# B&R Automation Studio project ABC_Pltzr
Automation Studio 4.2.4.149

## Configuration PPC70_24025GEN

CPU 4PPC70.101G-20W, AutomationRuntime D4.22, Build 4.1.2, Vc V4.24.0, Safety 0.0

### Hardware
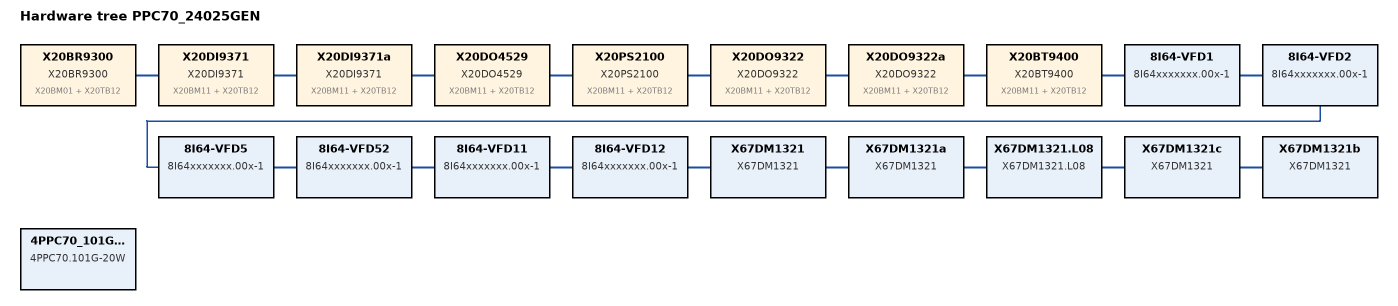
```
4PPC70_101G_20W : 4PPC70.101G-20W v1.2.0.0
  Connector IF1:
    ActivatePowerlink = 0
  Connector IF2:
    ActivateDevice = 1
    Mode = Manual
    InternetAddress = 192.168.1.100
    SubnetMask = 255.255.255.0
    InaNodeNumber = 1
    Vnc1
    VncVcObjectName1 = WSVGA
    VncAuthentication1 = 1
    VncPasswordViewOnly1 = v
    VncPasswordViewControl1 = 24025
    VncMaxConnections1 = 2
    VncRefreshRate1 = 250
  PermanentPvSize = 1000
  RemanentGlobalPvSize = 25000
  VolatileGlobalPvSize = 200000
  EnableUsbRemoteInstall = 1
  TimerDeviceType = SWIOTIMER
  Cyclic1Duration = 4000
  Cyclic1Tolerance = 4000
  Cyclic2Duration = 20000
  Cyclic2Tolerance = 20000
  Cyclic3Duration = 50000
  Cyclic3Tolerance = 50000
  Cyclic4Duration = 100000
  Cyclic4Tolerance = 100000
  Cyclic5Duration = 200000
  Cyclic5Tolerance = 200000
  Cyclic6Duration = 500000
  Cyclic6Tolerance = 500000
  Cyclic7Duration = 1000000
  Cyclic7Tolerance = 1000000
  Cyclic8Duration = 10000
  Cyclic8Tolerance = 30000000
  FtpUser1
  FtpUsername1 = abc
  FtpUserPassword1 = veVz20Da1KUF2Vww53L6omFNdzfk8lHY0HjcrjfOb/w=  // abc123
  FtpUserSalt1 = pyAcjG26
  FTPPath1 = 5
  FTPAccessRight1 = 0
  VcObjectName = WSVGA
  KeyMappingFile = VC\4PPC70_101G_20W.dis
8I64-VFD1 : 8I64xxxxxxx.00x-1 v1.3.8.1  [X2X1 -> X20BT9400.X2X1]
  FunctionModel = Standard
  Supervision = off
  enableIOLR = off
  enableDigitalOutput = off
  DigitalOutputMode01 = actionDO
  ACC = 1
  DEC = 1
  HSP = 900
  ITH = 28
  BFR = 1
  UNS = 460
  FRS = 600
  NCR = 28
  NSP = 1750
  COS = 80
  TFR = 900
  DO = 9
  BRA = 0
  BLC = 64
  BRT = 15
  BEN = 0
  BET = 15
8I64-VFD11 : 8I64xxxxxxx.00x-1 v1.3.8.1  [X2X1 -> 8I64-VFD52.X2X2]
  FunctionModel = Standard
  Supervision = off
  enableIOLR = off
  enableDigitalOutput = off
  DigitalOutputMode01 = actionDO
  DownloadParameters = yes
  ACC = 1
  DEC = 1
  HSP = 900
  ITH = 13
  FTD = 600
  BFR = 1
  UNS = 460
  FRS = 600
  NCR = 13
  NSP = 1750
  COS = 80
  TFR = 900
  DO = 9
  BRA = 0
  BLC = 64
  BRT = 5
  BEN = 0
  BET = 5
8I64-VFD12 : 8I64xxxxxxx.00x-1 v1.3.8.1  [X2X1 -> 8I64-VFD11.X2X2]
  FunctionModel = Standard
  Supervision = off
  enableIOLR = off
  enableDigitalOutput = off
  DigitalOutputMode01 = actionDO
  DownloadParameters = yes
  ACC = 1
  DEC = 200
  HSP = 900
  ITH = 13
  FTD = 600
  BFR = 1
  UNS = 460
  FRS = 600
  NCR = 13
  NSP = 1750
  COS = 80
  TFR = 900
  DO = 9
  BRA = 0
  BLC = 64
  BRT = 5
  BEN = 0
  BET = 5
8I64-VFD2 : 8I64xxxxxxx.00x-1 v1.3.8.1  [X2X1 -> 8I64-VFD1.X2X2]
  FunctionModel = Standard
  Supervision = off
  enableIOLR = off
  enableDigitalOutput = off
  DigitalOutputMode01 = actionDO
  DownloadParameters = yes
  ACC = 1
  DEC = 1
  HSP = 900
  BFR = 1
  UNS = 460
  FRS = 600
  NCR = 13
  NSP = 1750
  TFR = 900
  DO = 9
  BRA = 0
  BLC = 64
  BRT = 5
  BEN = 0
  BET = 5
8I64-VFD5 : 8I64xxxxxxx.00x-1 v1.3.8.1  [X2X1 -> 8I64-VFD2.X2X2]
  FunctionModel = Standard
  Supervision = off
  DownloadParameters = yes
  ACC = 1
  DEC = 1
  HSP = 900
  ITH = 13
  FTD = 600
  BFR = 1
  UNS = 460
  FRS = 600
  NCR = 13
  NSP = 1750
  COS = 80
  TFR = 900
  DE2 = 10
  BRA = 0
8I64-VFD52 : 8I64xxxxxxx.00x-1 v1.3.8.1  [X2X1 -> 8I64-VFD5.X2X2]
  FunctionModel = Standard
  Supervision = off
  enableIOLR = off
  enableDigitalOutput = off
  DigitalOutputMode01 = actionDO
  ACC = 1
  DEC = 1
  HSP = 900
  ITH = 13
  FTD = 600
  BFR = 1
  UNS = 460
  FRS = 600
  NCR = 13
  NSP = 1750
  COS = 80
  TFR = 900
  DO = 9
  INR = 0
  BRA = 0
  BLC = 64
  BRT = 1
  BEN = 0
  BET = 1
X20BM01 : X20BM01 v1.0.0.1
X20BM11 : X20BM11 v1.0.0.0  [X2X1 -> X20BM01.X2X2]
X20BM11a : X20BM11 v1.0.0.0  [X2X1 -> X20BM11.X2X2]
X20BM11b : X20BM11 v1.0.0.0  [X2X1 -> X20BM11a.X2X2]
X20BM11c : X20BM11 v1.0.0.0  [X2X1 -> X20BM11b.X2X2]
X20BM11d : X20BM11 v1.0.0.0  [X2X1 -> X20BM11c.X2X2]
X20BM11e : X20BM11 v1.0.0.0  [X2X1 -> X20BM11f.X2X2]
X20BM11f : X20BM11 v1.0.0.0  [X2X1 -> X20BM11d.X2X2]
X20BR9300 : X20BR9300 v1.0.2.6  [SS1 -> X20TB12.SS; SL -> X20BM01.SL1; X2X1 -> 4PPC70_101G_20W.IF5]
  Supervision = off
X20BT9400 : X20BT9400 v1.0.1.3  [SS1 -> X20TB12f.SS; SL -> X20BM11e.SL1]
  Supervision = off
X20DI9371 : X20DI9371 v1.0.1.2  [SS1 -> X20TB12a.SS; SL -> X20BM11.SL1]
  Supervision = off
X20DI9371a : X20DI9371 v1.0.1.2  [SS1 -> X20TB12b.SS; SL -> X20BM11a.SL1]
  Supervision = off
  InputFilter = 100
X20DO4529 : X20DO4529 v1.0.1.2  [SS1 -> X20TB12c.SS; SL -> X20BM11b.SL1]
  Supervision = off
X20DO9322 : X20DO9322 v1.0.3.0  [SS1 -> X20TB12e.SS; SL -> X20BM11d.SL1]
  Supervision = off
X20DO9322a : X20DO9322 v1.0.3.0  [SS1 -> X20TB12g.SS; SL -> X20BM11f.SL1]
  Supervision = off
X20PS2100 : X20PS2100 v1.0.3.0  [SS1 -> X20TB12d.SS; SL -> X20BM11c.SL1]
  Supervision = off
X20TB12 : X20TB12 v1.0.0.0
X20TB12a : X20TB12 v1.0.0.0
X20TB12b : X20TB12 v1.0.0.0
X20TB12c : X20TB12 v1.0.0.0
X20TB12d : X20TB12 v1.0.0.0
X20TB12e : X20TB12 v1.0.0.0
X20TB12f : X20TB12 v1.0.0.0
X20TB12g : X20TB12 v1.0.0.0
X67DM1321 : X67DM1321 v1.1.1.0  [X2X1 -> 8I64-VFD12.X2X2]
  Supervision = off
X67DM1321.L08 : X67DM1321.L08 v1.1.2.0  [X2X1 -> X67DM1321a.X2X2]
  Supervision = off
  Direction01 = output
  Direction02 = output
  Direction03 = output
  Direction04 = output
  Direction05 = output
  Direction06 = output
  Direction07 = output
  Direction08 = output
  Direction09 = output
  Direction10 = output
  Direction11 = output
  Direction12 = output
X67DM1321a : X67DM1321 v1.1.1.0  [X2X1 -> X67DM1321.X2X2]
  Supervision = off
  Direction01 = output
  Direction02 = output
  Direction03 = output
  Direction04 = output
X67DM1321b : X67DM1321 v1.1.1.0  [X2X1 -> X67DM1321c.X2X2]
  Supervision = off
X67DM1321c : X67DM1321 v1.1.1.0  [X2X1 -> X67DM1321.L08.X2X2]
  Supervision = off
  Direction01 = output
  Direction02 = output
```

## Configuration PPC70_JOB24025

### Task classes (Cpu.sw)
```
Cyclic#1:
  diofilter <- MachineControl.diofilter.prg
  simonly <- MachineControl.simonly.prg
  alarms <- MachineControl.alarms.prg
  messages <- MachineControl.messages.prg
  machCtrl <- MachineControl.machCtrl.prg
  machzero <- MachineControl.machzero.prg
  vfdControl <- MachineControl.vfdControl.prg
  safety <- MachineControl.safety.prg
  counter <- Simulation.counter.prg
  machmode <- MachineControl.machmode.prg
  caseturner <- MachineControl.caseturner.prg
  blades <- MachineControl.blades.prg
  rowforming <- MachineControl.rowforming.prg
  transtable <- MachineControl.transtable.prg
  retainbar <- MachineControl.retainbar.prg
  squaring <- MachineControl.squaring.prg
  elevator <- MachineControl.elevator.prg
  elevmove <- MachineControl.elevmove.prg
  palletinfe <- MachineControl.palletinfcv.prg
  palletdisc <- MachineControl.palletdischarge.prg
  infcvidle <- MachineControl.infcvidle.prg
  palletinfa <- MachineControl.palletinfauto.prg [disabled]
  animation <- MachineControl.animation.prg [disabled]
  palProc <- MachineControl.palProc.prg
  drycycle <- MachineControl.drycycle.prg [disabled]
  drycypal <- MachineControl.drycypal.prg [disabled]
Cyclic#4:
  X64param <- ParameterDownload.X64_S44_Download.X64param.prg [disabled]
  paiVFDX64 <- paiComponents.paiBnRVFD.paiVFDX64.prg
Cyclic#8:
  paiHmi <- paiComponents.paiTemplate.paiHMI.paiHmi.prg
  paiFS <- paiComponents.paiFileService.paiFS.prg
  paiMp <- paiComponents.paiMp.paiMp.prg
  paiFileDT <- paiComponents.paiMp.paiFileDT.prg
  paiUser <- paiComponents.paiUser.paiUser.prg
  appHmi <- MachineControl.appHmi.prg
  appDraw <- MachineControl.appDraw.prg
  appCfgRec <- appConfigAndRecipes.appCfgRec.prg
  paiPingSer <- paiComponents.paiPing.paiPingService.prg
  read_data <- paiComponents.LibAsUSB1_ST.read_data.prg [disabled]
VcDataObjects: WSVGA <- HMI.WSVGA.dob
Binaries: vccdt, vccbmp, vccline, vcfile, arial, vctcal, WSVGA02, vcrt, vcmgr, vccstr, vcbclass, vccbtn, vcgclass, vcdsint, vcchtml, vccpwd, vcshared, vccddbox, vccscale, arialbd, vcxml, vccnum, vccalarm, visvc, vccurl, vccslider, vcctext, vcpdsw, vcfntttf, vccovl, vccshape, ariblk, cour, vcctrend, vcclbox, vccpopup, vcdsloc, vcchspot, vcalarm, WSVGA01, WSVGA03, vcpdvnc, vcpkat, vcnet, vccdbox, vcpdi815, vcptelo, vcpdihd, vcpdi855, vcpfppc7, vcpk, Config_4, Config_3, Config_1, iomap, ashwd, Config_2, asfw, Config, arconfig, sysconf, vcpfar00
Libraries: sprintf2, bgringbuf, bglibas, standard, AsIecCon, Operator, asstring, brsystem, sys_lib, AsARCfg, AsUPS, FileIO, AsICMP, AsBrStr, MpCom, MpFile, MpRecipe, MpAlarm, dvframe, astime, visapi, arsvcreg, vcresman, dataobj, AsIOAcc, runtime, AsMem, AsMath, AsEPL, CSV_File, AsUSB
```

### Config_2.mpalarmbasic - 4PPC70_101G_20F005/mapp/Config_2.mpalarmbasic
```
Element gMpLinkMpAlarmBasic (Type=mpalarmbasic)
  mapp.Alarm.Factory:
    Reactions:
      Reaction[0]:
        Description = Example: Immediate Stop
  Alarms:
    UserAlarm:
      Alarms:
        Alarm[0]:
          ID = 0
          Description = Example: Temperature over Tolerance
          Reaction = 1
```

### Config_3.mprecipexml - 4PPC70_101G_20F005/mapp/Config_3.mprecipexml
```
Element gMpLinkMpRecipeXmlCustom1 (Type=mprecipexml)
```

## Configuration PPC70_Ver1

CPU 4PPC70.101G-20F005, AutomationRuntime D4.22, Build 4.1.2, Vc V4.22.0

### Task classes (Cpu.sw)
```
Cyclic#1:
  simonly <- MachineControl.simonly.prg
  alarms <- MachineControl.alarms.prg
  messages <- MachineControl.messages.prg
  machCtrl <- MachineControl.machCtrl.prg
  machzero <- MachineControl.machzero.prg
  vfdControl <- MachineControl.vfdControl.prg
  safety <- MachineControl.safety.prg
  counter <- Simulation.counter.prg
  machmode <- MachineControl.machmode.prg
  caseturner <- MachineControl.caseturner.prg
  blades <- MachineControl.blades.prg
  rowforming <- MachineControl.rowforming.prg
  transtable <- MachineControl.transtable.prg
  retainbar <- MachineControl.retainbar.prg
  squaring <- MachineControl.squaring.prg
  elevator <- MachineControl.elevator.prg
  elevmove <- MachineControl.elevmove.prg
  palletinfe <- MachineControl.palletinfcv.prg
  palletdisc <- MachineControl.palletdischarge.prg
  palletinfa <- MachineControl.palletinfauto.prg
  animation <- MachineControl.animation.prg [disabled]
  palProc <- MachineControl.palProc.prg
  drycycle <- MachineControl.drycycle.prg [disabled]
  drycypal <- MachineControl.drycypal.prg [disabled]
Cyclic#4:
  X64param <- ParameterDownload.X64_S44_Download.X64param.prg [disabled]
Cyclic#8:
  paiHmi <- paiComponents.paiTemplate.paiHMI.paiHmi.prg
  paiFS <- paiComponents.paiFileService.paiFS.prg
  paiMp <- paiComponents.paiMp.paiMp.prg
  paiFileDT <- paiComponents.paiMp.paiFileDT.prg
  paiUser <- paiComponents.paiUser.paiUser.prg
  appHmi <- MachineControl.appHmi.prg
  appDraw <- MachineControl.appDraw.prg
  appCfgRec <- appConfigAndRecipes.appCfgRec.prg
  paiPingSer <- paiComponents.paiPing.paiPingService.prg
VcDataObjects: WSVGA <- HMI.WSVGA.dob
Binaries: vccdt, vccbmp, vccline, vcfile, arial, vctcal, WSVGA02, vcrt, vcmgr, vccstr, vcbclass, vccbtn, vcgclass, vcdsint, vcchtml, vccpwd, vcshared, vccddbox, vccscale, arialbd, vcxml, vccnum, vccalarm, visvc, vccurl, vccslider, vcctext, vcpdsw, vcfntttf, vccovl, vccshape, ariblk, cour, vcctrend, vcclbox, vccpopup, vcdsloc, vcchspot, vcalarm, WSVGA01, WSVGA03, vcpdvnc, vcpkat, vcnet, vccdbox, vcpk, vcpfppc7, vcpdi855, vcpdihd, vcptelo, vcpdi815, vcpfar00, Config_4, Config_3, Config_1, iomap, ashwd, Config_2, asfw, Config, arconfig, sysconf
Libraries: sprintf2, bgringbuf, bglibas, standard, AsIecCon, Operator, asstring, brsystem, sys_lib, AsARCfg, AsUPS, FileIO, AsICMP, AsBrStr, MpCom, MpFile, MpRecipe, MpAlarm, dvframe, astime, visapi, arsvcreg, vcresman, dataobj, AsIOAcc, runtime, AsMem, AsMath, AsEPL, CSV_File
```

### IoMap.iom - 4PPC70_101G_20F005/IoMap.iom
```iecst
(*********************************************************************************
 * Copyright:
 * Author:    goran
 * Created:   August 31, 2015/10:10 PM
 *********************************************************************************
 * IO mapping
 *********************************************************************************)
VAR_CONFIG
	::gHWModules[1].ModuleOk AT %IX."X20BR9300".ModuleOk;
	::gHWModules[2].ModuleOk AT %IX."X20DI9371".ModuleOk;
	::gHWModules[3].ModuleOk AT %IX."X20DI9371a".ModuleOk;
	::gHWModules[4].ModuleOk AT %IX."X20DO4529".ModuleOk;
	::gHWModules[5].ModuleOk AT %IX."X20PS2100".ModuleOk;
	::gHWModules[6].ModuleOk AT %IX."X20DO9322".ModuleOk;
	gHWModules[7].ModuleOk AT %IX."X20DO9322a".ModuleOk;
	gHWModules[8].ModuleOk AT %IX."X20BT9400".ModuleOk;
	gHWModules[9].ModuleOk AT %IX."8I64-VFD1".ModuleOk;
	gHWModules[10].ModuleOk AT %IX."8I64-VFD2".ModuleOk;
	gHWModules[11].ModuleOk AT %IX."8I64-VFD4".ModuleOk;
	gHWModules[12].ModuleOk AT %IX."8I64-VFD11".ModuleOk;
	gHWModules[13].ModuleOk AT %IX."X67DM1321".ModuleOk;
	gHWModules[14].ModuleOk AT %IX."X67DM1321a".ModuleOk;
	gHWModules[15].ModuleOk AT %IX."X67DM1321.L08".ModuleOk;
	gHWModules[16].ModuleOk AT %IX."X67DM1321b".ModuleOk;
	gHWModules[17].ModuleOk AT %IX."X67DM1321.L08a".ModuleOk;
	::gMachineVFD[1].vfdIn.Status.ReadyToSwitchOn AT %IX."8I64-VFD1".ETAD_Input_Bool_00;
	::gMachineVFD[1].vfdIn.Status.SwitchedOn AT %IX."8I64-VFD1".ETAD_Input_Bool_01;
	::gMachineVFD[1].vfdIn.Status.OperationEnabled AT %IX."8I64-VFD1".ETAD_Input_Bool_02;
	::gMachineVFD[1].vfdIn.Status.FaultDetection AT %IX."8I64-VFD1".ETAD_Input_Bool_03;
	::gMachineVFD[1].vfdIn.Status.VoltageEnabled AT %IX."8I64-VFD1".ETAD_Input_Bool_04;
	::gMachineVFD[1].vfdIn.Status.QuickStop AT %IX."8I64-VFD1".ETAD_Input_Bool_05;
	::gMachineVFD[1].vfdIn.Status.SwitchOnDisabled AT %IX."8I64-VFD1".ETAD_Input_Bool_06;
	::gMachineVFD[1].vfdIn.Status.WarningAlarm AT %IX."8I64-VFD1".ETAD_Input_Bool_07;
	::gMachineVFD[1].vfdIn.Status.TargetReached AT %IX."8I64-VFD1".ETAD_Input_Bool_10;
	::gMachineVFD[1].vfdIn.Status.StopKey AT %IX."8I64-VFD1".ETAD_Input_Bool_14;
	::gMachineVFD[1].vfdIn.Status.Direction AT %IX."8I64-VFD1".ETAD_Input_Bool_15;
	::gMachineVFD[1].vfdIn.Status.Accelerating AT %IX."8I64-VFD1".ETI_Input_Bool_09;
	::gMachineVFD[1].vfdIn.Status.Decelerating AT %IX."8I64-VFD1".ETI_Input_Bool_10;
	::gMachineVFD[1].vfdIn.Status.FastStop AT %IX."8I64-VFD1".ETI_Input_Bool_12;
	::gMachineVFD[1].vfdIn.Status.CurrentVelocity AT %IW."8I64-VFD1".RFRD_Input;
	::gMachineVFD[1].vfdIn.Status.MotorTorque AT %IW."8I64-VFD1".OTR_Input;
	::gMachineVFD[1].vfdIn.Status.MotorCurrent AT %IW."8I64-VFD1".LCR_Input;
	::gMachineVFD[1].vfdIn.Status.DriveThermalState AT %IW."8I64-VFD1".THD_Input;
	::gMachineVFD[1].vfdIn.Status.MotorThermalState AT %IW."8I64-VFD1".THR_Input;
	::gMachineVFD[1].vfdIn.IO.LogicInput1 AT %IX."8I64-VFD1".IOLR_Input_Bool_00;
	::gMachineVFD[1].vfdIn.IO.LogicInput2 AT %IX."8I64-VFD1".IOLR_Input_Bool_01;
	::gMachineVFD[1].vfdIn.IO.LogicInput3 AT %IX."8I64-VFD1".IOLR_Input_Bool_02;
	::gMachineVFD[1].vfdIn.IO.LogicInput4 AT %IX."8I64-VFD1".IOLR_Input_Bool_03;
	::gMachineVFD[1].vfdIn.IO.Relay02State AT %IX."8I64-VFD1".IOLR_Input_Bool_09;
	::gMachineVFD[1].vfdIn.Fault.CurrentFault AT %IW."8I64-VFD1".ERRD_Input;
	::gMachineVFD[1].vfdIn.Fault.LastFault AT %IW."8I64-VFD1".LFT_Input;
	::gMachineVFD[1].vfdOut.Control.SwitchOn AT %QX."8I64-VFD1".CMDD_Output_Bool_00;
	::gMachineVFD[1].vfdOut.Control.DisableVoltage AT %QX."8I64-VFD1".CMDD_Output_Bool_01;
	::gMachineVFD[1].vfdOut.Control.QuickStop AT %QX."8I64-VFD1".CMDD_Output_Bool_02;
	::gMachineVFD[1].vfdOut.Control.EnableOperation AT %QX."8I64-VFD1".CMDD_Output_Bool_03;
	::gMachineVFD[1].vfdOut.Control.FaultReset AT %QX."8I64-VFD1".CMDD_Output_Bool_07;
	::gMachineVFD[1].vfdOut.Control.Direction AT %QX."8I64-VFD1".CMDD_Output_Bool_11;
	::gMachineVFD[1].vfdOut.Control.FastStop AT %QX."8I64-VFD1".CMDD_Output_Bool_12;
	::gMachineVFD[1].vfdOut.Control.VelocitySetpoint AT %QW."8I64-VFD1".LFRD_Output;
	::gMachineVFD[2].vfdIn.Status.ReadyToSwitchOn AT %IX."8I64-VFD2".ETAD_Input_Bool_00;
	::gMachineVFD[2].vfdIn.Status.SwitchedOn AT %IX."8I64-VFD2".ETAD_Input_Bool_01;
	::gMachineVFD[2].vfdIn.Status.OperationEnabled AT %IX."8I64-VFD2".ETAD_Input_Bool_02;
	::gMachineVFD[2].vfdIn.Status.FaultDetection AT %IX."8I64-VFD2".ETAD_Input_Bool_03;
	::gMachineVFD[2].vfdIn.Status.VoltageEnabled AT %IX."8I64-VFD2".ETAD_Input_Bool_04;
	::gMachineVFD[2].vfdIn.Status.QuickStop AT %IX."8I64-VFD2".ETAD_Input_Bool_05;
	::gMachineVFD[2].vfdIn.Status.SwitchOnDisabled AT %IX."8I64-VFD2".ETAD_Input_Bool_06;
	::gMachineVFD[2].vfdIn.Status.WarningAlarm AT %IX."8I64-VFD2".ETAD_Input_Bool_07;
	::gMachineVFD[2].vfdIn.Status.TargetReached AT %IX."8I64-VFD2".ETAD_Input_Bool_10;
	::gMachineVFD[2].vfdIn.Status.StopKey AT %IX."8I64-VFD2".ETAD_Input_Bool_14;
	::gMachineVFD[2].vfdIn.Status.Direction AT %IX."8I64-VFD2".ETAD_Input_Bool_15;
	::gMachineVFD[2].vfdIn.Status.Accelerating AT %IX."8I64-VFD2".ETI_Input_Bool_09;
	::gMachineVFD[2].vfdIn.Status.Decelerating AT %IX."8I64-VFD2".ETI_Input_Bool_10;
	::gMachineVFD[2].vfdIn.Status.FastStop AT %IX."8I64-VFD2".ETI_Input_Bool_12;
	::gMachineVFD[2].vfdIn.Status.CurrentVelocity AT %IW."8I64-VFD2".RFRD_Input;
	::gMachineVFD[2].vfdIn.Status.MotorTorque AT %IW."8I64-VFD2".OTR_Input;
	::gMachineVFD[2].vfdIn.Status.MotorCurrent AT %IW."8I64-VFD2".LCR_Input;
	::gMachineVFD[2].vfdIn.Status.DriveThermalState AT %IW."8I64-VFD2".THD_Input;
	::gMachineVFD[2].vfdIn.Status.MotorThermalState AT %IW."8I64-VFD2".THR_Input;
	::gMachineVFD[2].vfdIn.IO.LogicInput1 AT %IX."8I64-VFD2".IOLR_Input_Bool_00;
	::gMachineVFD[2].vfdIn.IO.LogicInput2 AT %IX."8I64-VFD2".IOLR_Input_Bool_01;
	::gMachineVFD[2].vfdIn.IO.LogicInput3 AT %IX."8I64-VFD2".IOLR_Input_Bool_02;
	::gMachineVFD[2].vfdIn.IO.LogicInput4 AT %IX."8I64-VFD2".IOLR_Input_Bool_03;
	::gMachineVFD[2].vfdIn.IO.Relay02State AT %IX."8I64-VFD2".IOLR_Input_Bool_09;
	::gMachineVFD[2].vfdIn.Fault.CurrentFault AT %IW."8I64-VFD2".ERRD_Input;
	::gMachineVFD[2].vfdIn.Fault.LastFault AT %IW."8I64-VFD2".LFT_Input;
	::gMachineVFD[2].vfdOut.Control.SwitchOn AT %QX."8I64-VFD2".CMDD_Output_Bool_00;
	::gMachineVFD[2].vfdOut.Control.DisableVoltage AT %QX."8I64-VFD2".CMDD_Output_Bool_01;
	::gMachineVFD[2].vfdOut.Control.QuickStop AT %QX."8I64-VFD2".CMDD_Output_Bool_02;
	::gMachineVFD[2].vfdOut.Control.EnableOperation AT %QX."8I64-VFD2".CMDD_Output_Bool_03;
	::gMachineVFD[2].vfdOut.Control.FaultReset AT %QX."8I64-VFD2".CMDD_Output_Bool_07;
	::gMachineVFD[2].vfdOut.Control.Direction AT %QX."8I64-VFD2".CMDD_Output_Bool_11;
	::gMachineVFD[2].vfdOut.Control.FastStop AT %QX."8I64-VFD2".CMDD_Output_Bool_12;
	::gMachineVFD[2].vfdOut.Control.VelocitySetpoint AT %QW."8I64-VFD2".LFRD_Output;
	::gMachineVFD[4].vfdIn.Status.ReadyToSwitchOn AT %IX."8I64-VFD4".ETAD_Input_Bool_00;
	::gMachineVFD[4].vfdIn.Status.SwitchedOn AT %IX."8I64-VFD4".ETAD_Input_Bool_01;
	::gMachineVFD[4].vfdIn.Status.OperationEnabled AT %IX."8I64-VFD4".ETAD_Input_Bool_02;
	::gMachineVFD[4].vfdIn.Status.FaultDetection AT %IX."8I64-VFD4".ETAD_Input_Bool_03;
	::gMachineVFD[4].vfdIn.Status.VoltageEnabled AT %IX."8I64-VFD4".ETAD_Input_Bool_04;
	::gMachineVFD[4].vfdIn.Status.QuickStop AT %IX."8I64-VFD4".ETAD_Input_Bool_05;
	::gMachineVFD[4].vfdIn.Status.SwitchOnDisabled AT %IX."8I64-VFD4".ETAD_Input_Bool_06;
	::gMachineVFD[4].vfdIn.Status.WarningAlarm AT %IX."8I64-VFD4".ETAD_Input_Bool_07;
	::gMachineVFD[4].vfdIn.Status.TargetReached AT %IX."8I64-VFD4".ETAD_Input_Bool_10;
	::gMachineVFD[4].vfdIn.Status.StopKey AT %IX."8I64-VFD4".ETAD_Input_Bool_14;
	::gMachineVFD[4].vfdIn.Status.Direction AT %IX."8I64-VFD4".ETAD_Input_Bool_15;
	::gMachineVFD[4].vfdIn.Status.Accelerating AT %IX."8I64-VFD4".ETI_Input_Bool_09;
	::gMachineVFD[4].vfdIn.Status.Decelerating AT %IX."8I64-VFD4".ETI_Input_Bool_10;
	::gMachineVFD[4].vfdIn.Status.FastStop AT %IX."8I64-VFD4".ETI_Input_Bool_12;
	::gMachineVFD[4].vfdIn.Status.CurrentVelocity AT %IW."8I64-VFD4".RFRD_Input;
	::gMachineVFD[4].vfdIn.Status.MotorTorque AT %IW."8I64-VFD4".OTR_Input;
	::gMachineVFD[4].vfdIn.Status.MotorCurrent AT %IW."8I64-VFD4".LCR_Input;
	::gMachineVFD[4].vfdIn.Status.DriveThermalState AT %IW."8I64-VFD4".THD_Input;
	::gMachineVFD[4].vfdIn.Status.MotorThermalState AT %IW."8I64-VFD4".THR_Input;
	::gMachineVFD[4].vfdIn.IO.LogicInput1 AT %IX."8I64-VFD4".IOLR_Input_Bool_00;
	::gMachineVFD[4].vfdIn.IO.LogicInput2 AT %IX."8I64-VFD4".IOLR_Input_Bool_01;
	::gMachineVFD[4].vfdIn.IO.LogicInput3 AT %IX."8I64-VFD4".IOLR_Input_Bool_02;
	::gMachineVFD[4].vfdIn.IO.LogicInput4 AT %IX."8I64-VFD4".IOLR_Input_Bool_03;
	::gMachineVFD[4].vfdIn.IO.Relay02State AT %IX."8I64-VFD4".IOLR_Input_Bool_09;
	::gMachineVFD[4].vfdIn.Fault.CurrentFault AT %IW."8I64-VFD4".ERRD_Input;
	::gMachineVFD[4].vfdIn.Fault.LastFault AT %IW."8I64-VFD4".LFT_Input;
	::gMachineVFD[4].vfdOut.Control.SwitchOn AT %QX."8I64-VFD4".CMDD_Output_Bool_00;
	::gMachineVFD[4].vfdOut.Control.DisableVoltage AT %QX."8I64-VFD4".CMDD_Output_Bool_01;
	::gMachineVFD[4].vfdOut.Control.QuickStop AT %QX."8I64-VFD4".CMDD_Output_Bool_02;
	::gMachineVFD[4].vfdOut.Control.EnableOperation AT %QX."8I64-VFD4".CMDD_Output_Bool_03;
	::gMachineVFD[4].vfdOut.Control.FaultReset AT %QX."8I64-VFD4".CMDD_Output_Bool_07;
	::gMachineVFD[4].vfdOut.Control.Direction AT %QX."8I64-VFD4".CMDD_Output_Bool_11;
	::gMachineVFD[4].vfdOut.Control.FastStop AT %QX."8I64-VFD4".CMDD_Output_Bool_12;
	::gMachineVFD[4].vfdOut.Control.VelocitySetpoint AT %QW."8I64-VFD4".LFRD_Output;
	::gMachineVFD[11].vfdIn.Status.ReadyToSwitchOn AT %IX."8I64-VFD11".ETAD_Input_Bool_00;
	::gMachineVFD[11].vfdIn.Status.SwitchedOn AT %IX."8I64-VFD11".ETAD_Input_Bool_01;
	::gMachineVFD[11].vfdIn.Status.OperationEnabled AT %IX."8I64-VFD11".ETAD_Input_Bool_02;
	::gMachineVFD[11].vfdIn.Status.FaultDetection AT %IX."8I64-VFD11".ETAD_Input_Bool_03;
	::gMachineVFD[11].vfdIn.Status.VoltageEnabled AT %IX."8I64-VFD11".ETAD_Input_Bool_04;
	::gMachineVFD[11].vfdIn.Status.QuickStop AT %IX."8I64-VFD11".ETAD_Input_Bool_05;
	::gMachineVFD[11].vfdIn.Status.SwitchOnDisabled AT %IX."8I64-VFD11".ETAD_Input_Bool_06;
	::gMachineVFD[11].vfdIn.Status.WarningAlarm AT %IX."8I64-VFD11".ETAD_Input_Bool_07;
	::gMachineVFD[11].vfdIn.Status.TargetReached AT %IX."8I64-VFD11".ETAD_Input_Bool_10;
	::gMachineVFD[11].vfdIn.Status.StopKey AT %IX."8I64-VFD11".ETAD_Input_Bool_14;
	::gMachineVFD[11].vfdIn.Status.Direction AT %IX."8I64-VFD11".ETAD_Input_Bool_15;
	::gMachineVFD[11].vfdIn.Status.Accelerating AT %IX."8I64-VFD11".ETI_Input_Bool_09;
	::gMachineVFD[11].vfdIn.Status.Decelerating AT %IX."8I64-VFD11".ETI_Input_Bool_10;
	::gMachineVFD[11].vfdIn.Status.FastStop AT %IX."8I64-VFD11".ETI_Input_Bool_12;
	::gMachineVFD[11].vfdIn.Status.CurrentVelocity AT %IW."8I64-VFD11".RFRD_Input;
	::gMachineVFD[11].vfdIn.Status.MotorTorque AT %IW."8I64-VFD11".OTR_Input;
	::gMachineVFD[11].vfdIn.Status.MotorCurrent AT %IW."8I64-VFD11".LCR_Input;
	::gMachineVFD[11].vfdIn.Status.DriveThermalState AT %IW."8I64-VFD11".THD_Input;
	::gMachineVFD[11].vfdIn.Status.MotorThermalState AT %IW."8I64-VFD11".THR_Input;
	::gMachineVFD[11].vfdIn.IO.LogicInput1 AT %IX."8I64-VFD11".IOLR_Input_Bool_00;
	::gMachineVFD[11].vfdIn.IO.LogicInput2 AT %IX."8I64-VFD11".IOLR_Input_Bool_01;
	::gMachineVFD[11].vfdIn.IO.LogicInput3 AT %IX."8I64-VFD11".IOLR_Input_Bool_02;
	::gMachineVFD[11].vfdIn.IO.LogicInput4 AT %IX."8I64-VFD11".IOLR_Input_Bool_03;
	::gMachineVFD[11].vfdIn.IO.Relay02State AT %IX."8I64-VFD11".IOLR_Input_Bool_09;
	::gMachineVFD[11].vfdIn.Fault.CurrentFault AT %IW."8I64-VFD11".ERRD_Input;
	::gMachineVFD[11].vfdIn.Fault.LastFault AT %IW."8I64-VFD11".LFT_Input;
	::gMachineVFD[11].vfdOut.Control.SwitchOn AT %QX."8I64-VFD11".CMDD_Output_Bool_00;
	::gMachineVFD[11].vfdOut.Control.DisableVoltage AT %QX."8I64-VFD11".CMDD_Output_Bool_01;
	::gMachineVFD[11].vfdOut.Control.QuickStop AT %QX."8I64-VFD11".CMDD_Output_Bool_02;
	::gMachineVFD[11].vfdOut.Control.EnableOperation AT %QX."8I64-VFD11".CMDD_Output_Bool_03;
	::gMachineVFD[11].vfdOut.Control.FaultReset AT %QX."8I64-VFD11".CMDD_Output_Bool_07;
	::gMachineVFD[11].vfdOut.Control.Direction AT %QX."8I64-VFD11".CMDD_Output_Bool_11;
	::gMachineVFD[11].vfdOut.Control.FastStop AT %QX."8I64-VFD11".CMDD_Output_Bool_12;
	::gMachineVFD[11].vfdOut.Control.VelocitySetpoint AT %QW."8I64-VFD11".LFRD_Output;
	::gMachineIO.din.Guard_DS1 AT %IX."X20DI9371".DigitalInput01;
	::gMachineIO.din.Guard_DS2 AT %IX."X20DI9371".DigitalInput02;
	::gMachineIO.din.Guard_DS3 AT %IX."X20DI9371".DigitalInput03;
	::gMachineIO.din.EStop_PB1 AT %IX."X20DI9371".DigitalInput07;
	::gMachineIO.din.EStop_PB2 AT %IX."X20DI9371".DigitalInput08;
	::gMachineIO.din.EStop_PB3 AT %IX."X20DI9371".DigitalInput09;
	::gMachineIO.din.EStop_PB4 AT %IX."X20DI9371".DigitalInput10;
	::gMachineIO.din.MotorOverloads_OL AT %IX."X20DI9371a".DigitalInput01;
	::gMachineIO.din.MCR AT %IX."X20DI9371a".DigitalInput02;
	::gMachineIO.din.CustomerDischargeEnable_CR6 AT %IX."X20DI9371a".DigitalInput03;
	gMachineIO.din.PalleteDischLightCurtain_OSSD1 AT %IX."X20DI9371a".DigitalInput04;
	gMachineIO.din.PalleteDischLightCurtain_OSSD2 AT %IX."X20DI9371a".DigitalInput05;
	gMachineIO.din.AirPressureSwitch_APS AT %IX."X20DI9371a".DigitalInput06;
	::gMachineIO.dout.MachineFaultBeacon_LT1 AT %QX."X20DO4529".DigitalOutput01;
	::gMachineIO.dout.MachineOkBeacon_LT2 AT %QX."X20DO4529".DigitalOutput02;
	::gMachineIO.dout.PalletLowSupplyBeacon_LT3 AT %QX."X20DO4529".DigitalOutput03;
	::gMachineIO.dout.CustomerMachineRunning_CR5 AT %QX."X20DO4529".DigitalOutput04;
	::gMachineIO.dout.LayerStopBarRaise_M3F AT %QX."X20DO9322".DigitalOutput03;
	::gMachineIO.dout.LayerStopBarLower_M3R AT %QX."X20DO9322".DigitalOutput04;
	::gMachineIO.dout.RowFormingRollers_M5 AT %QX."X20DO9322".DigitalOutput07;
	::gMachineIO.dout.ProductInfeedCV_M6 AT %QX."X20DO9322".DigitalOutput08;
	::gMachineIO.dout.PalletDispenserCV_M7 AT %QX."X20DO9322".DigitalOutput09;
	::gMachineIO.dout.PalletDispenserRaise_M8F AT %QX."X20DO9322".DigitalOutput10;
	::gMachineIO.dout.PalletDispenserLower_M8R AT %QX."X20DO9322".DigitalOutput11;
	::gMachineIO.dout.CustomerMachineRunning_CR4 AT %QX."X20DO9322".DigitalOutput12;
	::gMachineIO.din.ElevatorDetectPalletLayerLF_EE1 AT %IX."X67DM1321".DigitalInput01;
	::gMachineIO.din.ElevatorChainSlackLF_LS7 AT %IX."X67DM1321".DigitalInput03;
	::gMachineIO.din.ElevatorChainSlackRT_LS8 AT %IX."X67DM1321".DigitalInput04;
	::gMachineIO.din.TransferTableAtPallete_PR5 AT %IX."X67DM1321".DigitalInput05;
	::gMachineIO.din.TransferTableAtGrouping_PR6 AT %IX."X67DM1321".DigitalInput06;
	::gMachineIO.din.LayerStopBarUp_PR7 AT %IX."X67DM1321".DigitalInput07;
	::gMachineIO.din.LayerStopBarDown_PR8 AT %IX."X67DM1321".DigitalInput08;
	::gMachineIO.dout.SideSquaringExtend_SOL8A AT %QX."X67DM1321a".DigitalOutput01;
	::gMachineIO.dout.SideSquaringRetract_SOL8B AT %QX."X67DM1321a".DigitalOutput02;
	::gMachineIO.dout.CaseTurnerRaise_SOL2A AT %QX."X67DM1321.L08".DigitalOutput01;
	::gMachineIO.dout.CaseTurnerLower_SOL2B AT %QX."X67DM1321.L08".DigitalOutput02;
	::gMachineIO.dout.BladeStop1Up_SOL3A AT %QX."X67DM1321.L08".DigitalOutput03;
	::gMachineIO.dout.BladeStop1Dw_SOL3B AT %QX."X67DM1321.L08".DigitalOutput04;
	::gMachineIO.din.ProductAtInfeed_EE2 AT %IX."X67DM1321.L08".DigitalInput13;
	::gMachineIO.din.RowTooLong_EE8 AT %IX."X67DM1321.L08".DigitalInput14;
	::gMachineIO.din.RowPusherReturned_PR11 AT %IX."X67DM1321.L08".DigitalInput15;
	::gMachineIO.din.RowPusherAtElevator_PR13 AT %IX."X67DM1321.L08".DigitalInput16;
	::gMachineIO.din.ElevatorFullUp_PR1 AT %IX."X67DM1321b".DigitalInput01;
	::gMachineIO.din.ElevatorFullDown_PR2 AT %IX."X67DM1321b".DigitalInput02;
	::gMachineIO.din.ElevatorAtGroupingLower_PR3 AT %IX."X67DM1321b".DigitalInput03;
	::gMachineIO.din.ElevatorAtGroupingRaise_PR4 AT %IX."X67DM1321b".DigitalInput04;
	::gMachineIO.din.ElevatorStopBlockLF_PR33 AT %IX."X67DM1321b".DigitalInput05;
	::gMachineIO.din.ElevatorStopBlockRT_PR34 AT %IX."X67DM1321b".DigitalInput06;
	::gMachineIO.din.PalletAtMachine_EE12 AT %IX."X67DM1321b".DigitalInput07;
	::gMachineIO.din.PalletAtDischarge_EE16 AT %IX."X67DM1321b".DigitalInput08;
	::gMachineIO.din.PalletClawsAtTop_PR14 AT %IX."X67DM1321.L08a".DigitalInput01;
	::gMachineIO.din.PalletClawsAtMiddleLow_PR15 AT %IX."X67DM1321.L08a".DigitalInput02;
	::gMachineIO.din.PalletClawsAtMiddleHi_PR15A AT %IX."X67DM1321.L08a".DigitalInput03;
	::gMachineIO.din.PalletClawsAtBottom_PR16 AT %IX."X67DM1321.L08a".DigitalInput04;
	::gMachineIO.din.PalletClawsClosedRT_PR18 AT %IX."X67DM1321.L08a".DigitalInput05;
	::gMachineIO.din.PalletClawsClosedLF_PR20 AT %IX."X67DM1321.L08a".DigitalInput06;
	::gMachineIO.din.PalletDispenserLowSupply_EE7 AT %IX."X67DM1321.L08a".DigitalInput07;
	::gMachineIO.dout.PalletClawsClose_SOL7A AT %QX."X67DM1321.L08a".DigitalOutput08;
	::gMachineIO.dout.PalletClawsOpen_SOL7B AT %QX."X67DM1321.L08a".DigitalOutput09;
	::gMachineIO.din.PalletDispenserChainSlack_PR21 AT %IX."X67DM1321.L08a".DigitalInput10;
	::gMachineIO.din.PalletDownOnDispenserCV_EE9 AT %IX."X67DM1321.L08a".DigitalInput11;
	::gMachineIO.dout.AirDump_SOL0 AT %QX."X20DO9322a".DigitalOutput01;
	::gMachineIO.dout.SheetInserterToMagazine AT %QX."X20DO9322a".DigitalOutput02;
	gMachineIO.din.PalletMagazineControl_SS2 AT %IX."X20DI9371a".DigitalInput07;
	gMachineIO.dout.BladeStop2Up_SOL4A  AT %QX."X67DM1321.L08".DigitalOutput05;
	gMachineIO.dout.BladeStop3Up_SOL5A  AT %QX."X67DM1321.L08".DigitalOutput07;
	gMachineIO.dout.BladeStop4Up_SOL6A  AT %QX."X67DM1321.L08".DigitalOutput09;
	gMachineIO.dout.BladeStop5Up_SOL13A  AT %QX."X67DM1321.L08".DigitalOutput11;
	gMachineIO.dout.BladeStop2Dw_SOL4B  AT %QX."X67DM1321.L08".DigitalOutput06;
	gMachineIO.dout.BladeStop3Dw_SOL5B  AT %QX."X67DM1321.L08".DigitalOutput08;
	gMachineIO.dout.BladeStop4Dw_SOL6B  AT %QX."X67DM1321.L08".DigitalOutput10;
	gMachineIO.dout.BladeStop5Dw_SOL13B  AT %QX."X67DM1321.L08".DigitalOutput12;
END_VAR
```

## Configuration testsim

### Task classes (Cpu.sw)
```
Cyclic#8:
  simonly <- Simulation.simonly.prg [disabled]
  paiPingSer <- paiComponents.paiPing.paiPingService.prg
  paiUser <- paiComponents.paiUser.paiUser.prg
  paiFileDT <- paiComponents.paiMp.paiFileDT.prg
  paiMp <- paiComponents.paiMp.paiMp.prg
  paiHmi <- paiComponents.paiTemplate.paiHMI.paiHmi.prg
  appCfgRec <- appConfigAndRecipes.appCfgRec.prg
  paiFS <- paiComponents.paiFileService.paiFS.prg
VcDataObjects: paXGA <- paiComponents.paiTemplate.paiHMI.paiScreens.paXGA.dob
Binaries: vcpkat, vccshape, vcctext, vcrt, vcchspot, vccstr, vcresman, vcfile, vcdsint, vcpdsw, arial, vcmgr, visvc, vcdsloc, vcfntttf, vccovl, vctcal, arialbd, vcalarm, vccnum, vcpdvnc, vcshared, vcpfar00, vccbtn, vcgclass, vcbclass, vcnet, vccslider, vccddbox, vccbmp, vccpopup, vcchtml, vcxml, vccpwd, vccalarm, vccurl, ariblk, cour, vccline, vcclbox, paXGA03, paXGA02, paXGA01, vcctrend, vccdt, vccscale, sysconf, ashwd, asfw, iomap, arconfig, Config_1, Config_2, Config, vccbar, visqc102, visqc101, visqc103, courbd, arialbi, visqc201, visqc202, visqc203, Visu01, Visu03, Visu02, Visu202, Visu201, Visu203
Libraries: AsUDP, astime, runtime, AsUPS, dvframe, dataobj, visapi, AsIecCon, standard, AsBrStr, sprintf2, bgringbuf, bglibas, FileIO, sys_lib, asarcfg, asicmp, asstring, arsvcreg, brsystem, MpCom, MpFile, MpRecipe, MpAlarm
```

### Cpu.per - PLC1/Cpu.per
```iecst
(********************************************************************
 * COPYRIGHT -- HP
 ********************************************************************
 * File: Cpu.per
 * Author: goran
 * Created: January 31, 2013
 ********************************************************************
 * Declaration of permanent variables
 ********************************************************************)
VAR_CONFIG
	gREMMEMPrefix AT %MD0; (* *)
	gHmiRemMem AT %M4; (* *)
	gREMMEMPostfix AT %MD104; (* *)
END_VAR
```

## Logical view

Binary libraries used (declarations not repeated): AsIecCon, Operator, DataObj, dvframe, asstring, EthSock, brsystem, sys_lib, Ethernet, standard, Visapi, AsUDP, astime, runtime, AsARCfg, AsUPS, FileIO, AsTCP, AsICMP, AsBrStr, AsIOAcc, AsMem, AsMath, AsEPL, MpCom, MpFile, MpRecipe 1.20.3, MpAlarm, AsUSB, sprintf2, bgringbuf


### Package Logical/paiComponents - pai Components and Libraries

### _X_bgftpclient.c
```c
#include <bur/plc.h>
#include <bur/plctypes.h>
#include <ethernet.h>
#include <ethsock.h>
#include <asstring.h>
#include <brsystem.h>
#include <sys_lib.h>

#include "bgstatemachine.h"
#include "bgstring.h"
#include "bgFtpClient.h"

#include "bgdebug.h"

#include "bgstatemachine.c"
#include "bgstring.c"

/*
History:
9/11/2005
- added support for receiving large files over ftp
- added error event for user ftp commands:
int bgFtpClientCmd<CmdName>OnError(bgFtpClient_typ *p);

*/

void ftpClientConnect(bgFtpClient_typ *p, int msgId);
int ftpClientConnectOnDone(bgFtpClient_typ *p);
int ftpClientConnectOnError(bgFtpClient_typ *p);

void ftpClientLogin(bgFtpClient_typ *p, int msgId);
int ftpClientLoginOnDone(bgFtpClient_typ *p);
int ftpClientLoginOnError(bgFtpClient_typ *p);

void ftpClientLogout(bgFtpClient_typ *p, int msgId);
int ftpClientLogoutOnDone(bgFtpClient_typ *p);
int ftpClientLogoutOnError(bgFtpClient_typ *p);

void ftpClientCmdGetFile(bgFtpClient_typ *p);

void ftpClientCmdList(bgFtpClient_typ *p);

void ftpClientCmdPwd(bgFtpClient_typ *p);

void ftpClientCmdCwd(bgFtpClient_typ *p);

void ftpClientDataServer(bgFtpClient_typ *p, int msgId);
int ftpClientDataServerOnError(bgFtpClient_typ *p);
int ftpClientDataServerOnDone(bgFtpClient_typ *p);

void ftpClientSingleCmdInit(bgFtpClient_typ *p, char *cmd, char *expectedServerResponse);
void ftpClientSingleCmd(bgFtpClient_typ *p);
int ftpClientSingleCmdOnError(bgFtpClient_typ *p);
int ftpClientSingleCmdOnDone(bgFtpClient_typ *p);

void ftpClientExecuteUserCmd_cyclic(bgFtpClient_typ *p);

int ftpClientCmdMultiOnDone(bgFtpClient_typ *p, int cmdId);
int ftpClientMultiCmdOnError(bgFtpClient_typ *p, int cmdId);
int ftpClientCmdCheckServerResponseCode(bgFtpClient_typ *p);

void ftpClientInitDataPort(bgFtpClient_typ *p);
void swapBytesInShort(unsigned short *value);
void setSocketAddressData(ETH_sockaddr_typ *adrData, char *hostIpAddressString, unsigned short hostPort);
void ftpClientGetResponse(bgFtpClient_typ *p);

void ftpClientCmdTextPort(bgFtpClient_typ *p, char *textBuffer);
void ftpClientMutliStateCmdErrorLog(bgFtpClient_typ *p);

int ftpClientIncrDataPort(bgFtpClient_typ *p);

/*
########################################################################################
========================================================================================
- FTP client protocol main state machine
- must be executed as a cyclic task (<=100ms)
- protocol implemenation uses nested state machines (several levels deep)
- FTP functions such as: connect, disconnect, login, logout and different FTP commands
are all implemented as state machines
*/
void bgFtpClientCyclic(bgFtpClient_typ *p, int msgId)
{
bgStateMachine_typ *psm = &p->smFtp;

	/*FTP client top level state machine*/
	switch( bgSMCyclic(psm) ){
		case 1:
          	/*idle; monitor user connection request flag*/
			bgSMSetStateName(psm, "Idle");

          	if(p->user.connectRequest){
	            p->user.connectRequest = 0;
	            p->user.disconnectRequest = 0;
				bgSMSetNextState(psm, bgSMGetState(psm) + 1);
          	}
		break;
		case 2:
			/*connect to FTP server*/
			bgSMSetStateName(psm, "Connect");

			if(bgSMIsStateInit(psm)){
				ftpClientConnect(p, BGSM_MSGID_INIT);
			}

			ftpClientConnect(p, BGSM_MSGID_CYCLIC);

			/*check if we are connected to FTP server*/
			if( p->isConnected ){
				bgSMSetNextState(psm, bgSMGetState(psm) + 1);
			}

			if(	ftpClientConnectOnError(p)){
                ERRxwarning(USER_ERROR_FTP, 1, "ftpClient-Err-socket()");
				bgSMRaiseError(psm, "error in lower level SM", 1, 0);
            }
		break;
		case 3:
			/*login*/
			bgSMSetStateName(psm, "Login");

			if(bgSMIsStateInit(psm)){
				ftpClientLogin(p, BGSM_MSGID_INIT);
			}

			ftpClientLogin(p, BGSM_MSGID_CYCLIC);

			/*check if we are looged-in*/
			if(p->isLoggedIn){
				p->userState = 0;
				bgSMSetNextState(psm, bgSMGetState(psm) + 1);
			}
			if(ftpClientLoginOnError(p)){
                ERRxwarning(USER_ERROR_FTP, 1, "ftpClient-Err-login()");
				bgSMRaiseError(psm, "error in lower level SM", 0, 0);
            }
		break;
		case 4:
            /*connected & logged-in -> normal operational state*/
			bgSMSetStateName(psm, "Ready");

			/*monitor requests & execute FTP commands*/
			ftpClientExecuteUserCmd_cyclic(p);

			/*terminate if socket error detected*/
			if(p->cmdError == ERR_SOCKET){
				bgSMSetNextState(psm, bgSMGetState(psm) + 1);
			}

			if(p->test){
				p->test = 0;
				ftpClientGetResponse(p);
			}

            /*monitor user disconnect request*/
            /*NOTE: upon receiving request, make sure to wait that FTP command in progress completes!*/

			/*disconnect allowed only after command completes*/
            if(p->user.disconnectRequest && !p->userState){
                p->user.connectRequest = 0;
                p->user.disconnectRequest = 0;
				bgSMSetNextState(psm, bgSMGetState(psm) + 1);
            }
		break;
		case 5:
            /*logout*/
			bgSMSetStateName(psm, "Logout");

			if(bgSMIsStateInit(psm)){
				ftpClientLogout(p, BGSM_MSGID_INIT);
			}

			ftpClientLogout(p, BGSM_MSGID_CYCLIC);

			/*chech if we are logged out*/
			if(!p->isLoggedIn){
				bgSMSetNextState(psm, bgSMGetState(psm) + 1);
			}

			if(ftpClientLogoutOnError(p)){
                ERRxwarning(USER_ERROR_FTP, 1, "ftpClient-Err-socket()");
				bgSMRaiseError(psm, "error in lower level SM", 0, 0);
            }
		break;
		case 6:
			bgSMSetStateName(psm, "Close CMD socket");
            /*normal operation; close socket*/
			bgSMRaiseDone(psm, 0);
		break;
		default:
			/*unhandled state*/
			bgSMRaiseError(psm, "unknown state", 0, bgSMGetState(psm));
		break;
	}

	if(bgSMOnDone(psm)){
		/*error state; socket closing is needed*/
		close(p->sock);

		p->isConnected = 0;

		bgSMSetNextState(psm, 1);
	}

	if(bgSMOnError(psm)){
		/*check if socket close needed or not?*/
		if( !bgSMGetErrorId(psm) )
			close(p->sock);

		p->isConnected = 0;
		p->cmdError = 1;
		bgSMSetNextState(psm, 1);
	}
}
/*
########################################################################################
	 INDIVIDUAL FTP COMMANDS
- each individual FTP command has following USER level interface methods:
	ftpClientCmd<Name>Init()
		- start command execution; pass-in user parameters; init cmd state machine
	ftpClientCmd<Name>OnDone()
		- monitor cmd completion (0-not complete; 1-complete)

- each command also has core implemenation (not used or called by the user)
	ftpClientCmd<Name>()

- FTP commands such as: PWD, CWD, PUT, GET, DIR are multi-level commands: it usually takes
several primitive FTP commands (i.e. PORT, TYPE, RETR etc) to complete one FTP command

########################################################################################
*/

/*
========================================================================================
- state machine that handles execution of individual, multi-level FTP commands
- FTP client executes one Multi-level command at the time
*/
void ftpClientExecuteUserCmd_cyclic(bgFtpClient_typ *p)
{
	/*execute user commands*/
	switch(p->userState){
	/*idle*/
        case 0:
        break;
        case 1:
        break;
        case 2:
            ftpClientCmdList(p);
        break;
        case 4:
            ftpClientCmdPwd(p);
        break;
        case 6:
            ftpClientCmdGetFile(p);
        break;
        case 8:
            ftpClientCmdCwd(p);
        break;
        default:
            p->userState = 0;
        break;
	}

}

/*
========================================================================================
FTP Command Implementation:
GetFile
*/
void bgFtpClientCmdGetFileInit(bgFtpClient_typ *p, char *fileName, char* buffer, int bufferLength)
{
    /*select command to execute*/
	p->userState = 6;

	/*pass command parameters*/
	p->user.dataBuffer = buffer;
	p->user.dataBufferLength = bufferLength;
	brsstrcpy((UDINT)&p->user.fileName[0], (UDINT)fileName);

    /*start command execution*/
	bgSMReset(&p->smFtpMultiCmd);
}

int bgFtpClientCmdGetFileOnDone(bgFtpClient_typ *p)
{
	return ftpClientCmdMultiOnDone(p, 6);
}

int bgFtpClientCmdGetFileOnError(bgFtpClient_typ *p)
{
	return ftpClientMultiCmdOnError(p, 6);
}

void ftpClientCmdGetFile(bgFtpClient_typ *p)
{
char cmdText[256];
bgStateMachine_typ *psm = &p->smFtpMultiCmd;

	/*FTP client multi level command state machine*/
	switch( bgSMCyclic(psm) ){
		case 1:
          	/*idle - monitor user connection request flag*/
			bgSMSetStateName(psm, "GetFile-InitDataSocket");

			if( bgSMIsStateInit(psm) ){
				/*generate port number to use*/
				ftpClientIncrDataPort(p);
				/*init Data transport socket*/
	            ftpClientDataServer(p, BGSM_MSGID_INIT);
			}

			/*wait for ready msg from the DataServer*/
            if( p->isDataPortReady ){
				bgSMSetNextState(psm, bgSMGetState(psm) + 1);
            }
/*TODO: timeout*/
		break;
		case 2:
    		/*PORT command: "PORT 192,168,1,6,0,20<CR><LF>"*/
			bgSMSetStateName(psm, "GetFile-PORT");
			if(bgSMIsStateInit(psm)){
	    		/*send command*/
	            ftpClientCmdTextPort(p, &cmdText[0]);

	    		ftpClientSingleCmdInit(p, &cmdText[0], "2??");
			}

    		/*recv cmd response*/
    		ftpClientSingleCmd(p);
			if(ftpClientSingleCmdOnDone(p)){
				bgSMSetNextState(psm, bgSMGetState(psm) + 1);
			}
			if(ftpClientSingleCmdOnError(p)){
				bgSMRaiseError(psm, "error in lower level SM", 0, 0);
			}
		break;
		case 3:
    		/*TYPE command: "TYPE I<CR><LF>"*/
			bgSMSetStateName(psm, "GetFile-TYPE");
			if(bgSMIsStateInit(psm)){
	    		/*send command*/
	    		ftpClientSingleCmdInit(p, "TYPE I", "2??");
			}

    		/*recv cmd response*/
    		ftpClientSingleCmd(p);
			if(ftpClientSingleCmdOnDone(p)){
				bgSMSetNextState(psm, bgSMGetState(psm) + 1);
			}

			if(ftpClientSingleCmdOnError(p)){
				bgSMRaiseError(psm, "error in lower level SM", 0, 0);
			}
		break;
		case 4:
    		/*RETR command: "RETR<CR><LF>""*/
			bgSMSetStateName(psm, "GetFile-RETR");
			if(bgSMIsStateInit(psm)){
	    		/*send command*/
	    		/*send command*/
	    		brsstrcpy((UDINT)&cmdText[0], (UDINT)"RETR ");
	    		brsstrcat((UDINT)&cmdText[0], (UDINT)&p->user.fileName[0]);
	    		ftpClientSingleCmdInit(p, &cmdText[0], "2??");
			}

    		/*recv cmd response*/
    		ftpClientSingleCmd(p);
			if(ftpClientSingleCmdOnDone(p)){
				/*notify data port server that the response is comming*/
				ftpClientDataServer(p, 2);
				bgSMSetNextState(psm, bgSMGetState(psm) + 1);
			}

			if(ftpClientSingleCmdOnError(p)){
				bgSMRaiseError(psm, "error in lower level SM", 0, 0);
				/*close data server port*/
				ftpClientDataServer(p, 3);
			}
		break;
        case 5:
			bgSMSetStateName(psm, "GetFile-DATASRVR active");
        break;
		default:
			/*unhandled state*/
			bgSMRaiseError(psm, "unknown state", 0, bgSMGetState(psm));
		break;
	}

	if(bgSMOnError(psm)){
		p->isErrorMultiCmd = p->userState;
		p->userState = 0;
		return;
	}

	ftpClientDataServer(p, BGSM_MSGID_CYCLIC);

	if(ftpClientDataServerOnDone(p)){
		p->isDoneMultiCmd = p->userState;
		p->userState = 0;
	}

	if(ftpClientDataServerOnError(p)){
		p->isErrorMultiCmd = p->userState;
		p->userState = 0;
	}

}
/*
========================================================================================
FTP Command Implementation:
List (dir)
*/
void bgFtpClientCmdListInit(bgFtpClient_typ *p, char *buffer, int bufferLength)
{
    /*select command to execute*/
	p->userState = 2;

	/*pass command parameters*/
	p->user.dataBuffer = buffer;
	p->user.dataBufferLength = bufferLength;

    /*start command execution*/
	bgSMReset(&p->smFtpMultiCmd);
}

int bgFtpClientCmdListOnDone(bgFtpClient_typ *p)
{
	return ftpClientCmdMultiOnDone(p, 2);
}

int bgFtpClientCmdListOnError(bgFtpClient_typ *p)
{
	return ftpClientMultiCmdOnError(p, 2);

}

void ftpClientCmdList(bgFtpClient_typ *p)
{
char cmdText[64];
bgStateMachine_typ *psm = &p->smFtpMultiCmd;

	/*FTP client multi level command state machine*/
	switch( bgSMCyclic(psm) ){
		case 1:
          	/*idle - monitor user connection request flag*/
			bgSMSetStateName(psm, "List-InitDataSocket");

			if( bgSMIsStateInit(psm) ){
				/*generate port number to use*/
				ftpClientIncrDataPort(p);
				/*init Data transport socket*/
	            ftpClientDataServer(p, BGSM_MSGID_INIT);
			}

			/*wait for ready msg from the DataServer*/
            if( p->isDataPortReady ){
				bgSMSetNextState(psm, bgSMGetState(psm) + 1);
            }
/*TODO: timeout*/
		break;
		case 2:
    		/*PORT command: "PORT 192,168,1,6,0,20<CR><LF>"*/
			bgSMSetStateName(psm, "List-PORT");
			if(bgSMIsStateInit(psm)){
	    		/*send command*/
	            ftpClientCmdTextPort(p, &cmdText[0]);

	    		ftpClientSingleCmdInit(p, &cmdText[0], "2??");
			}

    		/*recv cmd response*/
    		ftpClientSingleCmd(p);
			if(ftpClientSingleCmdOnDone(p)){
				bgSMSetNextState(psm, bgSMGetState(psm) + 1);
			}
			if(ftpClientSingleCmdOnError(p)){
				bgSMRaiseError(psm, "error in lower level SM", 0, 0);
			}
		break;
		case 3:
    		/*TYPE command: "TYPE I<CR><LF>"*/
			bgSMSetStateName(psm, "List-TYPE");
			if(bgSMIsStateInit(psm)){
	    		/*send command*/
	    		ftpClientSingleCmdInit(p, "TYPE I", "2??");
			}

    		/*recv cmd response*/
    		ftpClientSingleCmd(p);
			if(ftpClientSingleCmdOnDone(p)){
				bgSMSetNextState(psm, bgSMGetState(psm) + 1);
			}

			if(ftpClientSingleCmdOnError(p)){
				bgSMRaiseError(psm, "error in lower level SM", 0, 0);
			}
		break;
		case 4:
    		/*LIST command: "LIST<CR><LF>""*/
			bgSMSetStateName(psm, "List-List");
			if(bgSMIsStateInit(psm)){
	    		/*send command*/
	    		ftpClientSingleCmdInit(p, "LIST", "2??");
			}

    		/*recv cmd response*/
    		ftpClientSingleCmd(p);
			if(ftpClientSingleCmdOnDone(p)){
				/*notify data port server that the response is comming*/
				ftpClientDataServer(p, 2);
				bgSMSetNextState(psm, bgSMGetState(psm) + 1);
			}

			if(ftpClientSingleCmdOnError(p)){
				/*close data server port*/
				ftpClientDataServer(p, 3);
				bgSMRaiseError(psm, "error in lower level SM", 0, 0);
			}
		break;
        case 5:
			bgSMSetStateName(psm, "List-DATASRVR active");
        break;
		default:
			/*unhandled state*/
			bgSMRaiseError(psm, "unknown state", 0, bgSMGetState(psm));
		break;
	}

	if(bgSMOnError(psm)){
		p->isErrorMultiCmd = p->userState;
		p->userState = 0;
		return;
	}

	ftpClientDataServer(p, BGSM_MSGID_CYCLIC);

	if(ftpClientDataServerOnDone(p)){
		p->isDoneMultiCmd = p->userState;
		p->userState = 0;
	}

	if(ftpClientDataServerOnError(p)){
		p->isErrorMultiCmd = p->userState;
		p->userState = 0;
	}
}
/*
========================================================================================
FTP Command Implementation:
Pwd (Print Working Directory)
*/
void bgFtpClientCmdPwdInit(bgFtpClient_typ *p, char *buffer, int bufferLength)
{
    /*select command to execute*/
	p->userState = 4;

	/*pass command parameters*/
	p->user.dataBuffer = buffer;
	p->user.dataBufferLength = bufferLength;

    /*start command execution*/
	bgSMReset(&p->smFtpMultiCmd);
}

int bgFtpClientCmdPwdOnDone(bgFtpClient_typ *p)
{
	return ftpClientCmdMultiOnDone(p, 4);
}

int bgFtpClientCmdPwdOnError(bgFtpClient_typ *p)
{
	return ftpClientMultiCmdOnError(p, 4);

}

void ftpClientCmdPwd(bgFtpClient_typ *p)
{
bgStateMachine_typ *psm = &p->smFtpMultiCmd;

	/*FTP client multi level command state machine*/
	switch( bgSMCyclic(psm) ){
		case 1:
    		/*XPWD command: "XPWD<CR><LF>"*/
			bgSMSetStateName(psm, "PWD");
			if(bgSMIsStateInit(psm)){
	    		/*send command*/
	    		ftpClientSingleCmdInit(p, "PWD", "2??");
			}

    		/*recv cmd response*/
    		ftpClientSingleCmd(p);

			if(ftpClientSingleCmdOnDone(p)){
				/*copy response strig into the user supplied buffer*/
				brsstrcpy((UDINT)p->user.dataBuffer, (UDINT)p->responseList.items[0]);
				bgSMRaiseDone(psm, 0);
			}

			if(ftpClientSingleCmdOnError(p)){
				bgSMRaiseError(psm, "got lower SM error", 0, 0);
			}
		break;
		default:
			/*unhandled state*/
			bgSMRaiseError(psm, "unknown state", 0, bgSMGetState(psm));
		break;
	}

	if(bgSMOnError(psm)){
		p->userState = 0;
	}

	if(bgSMOnDone(psm)){
		p->isDoneMultiCmd = p->userState;
		p->userState = 0;
	}

}
/*
========================================================================================
FTP Command Implementation:
Cwd (Change Working Directory)
*/
void bgFtpClientCmdCwdInit(bgFtpClient_typ *p, char *fileName, char *buffer, int bufferLength)
{
    /*select command to execute*/
	p->userState = 8;

	/*pass command parameters*/
	p->user.dataBuffer = buffer;
	p->user.dataBufferLength = bufferLength;
	brsstrcpy((UDINT)&p->user.fileName[0], (UDINT)fileName);

    /*start command execution*/
	bgSMReset(&p->smFtpMultiCmd);

}

int bgFtpClientCmdCwdOnDone(bgFtpClient_typ *p)
{
	return ftpClientCmdMultiOnDone(p, 8);
}

int bgFtpClientCmdCwdOnError(bgFtpClient_typ *p)
{
	return ftpClientMultiCmdOnError(p, 8);

}

void ftpClientCmdCwd(bgFtpClient_typ *p)
{
char cmdText[255];

bgStateMachine_typ *psm = &p->smFtpMultiCmd;

	/*FTP client multi level command state machine*/
	switch( bgSMCyclic(psm) ){
		case 1:
    		/*XPWD command: "CWD <fileName><CR><LF>"*/
			bgSMSetStateName(psm, "CWD");
			if(bgSMIsStateInit(psm)){
	    		/*send command: "CWD <fileName><CR><LF>"*/
	    		brsstrcpy((UDINT)&cmdText[0], (UDINT)"CWD ");
	    		brsstrcat((UDINT)&cmdText[0], (UDINT)&p->user.fileName[0]);
	    		ftpClientSingleCmdInit(p, &cmdText[0], "2??");
			}

    		/*recv cmd response*/
    		ftpClientSingleCmd(p);

			if(ftpClientSingleCmdOnDone(p)){
				/*copy response strig into the user supplied buffer*/
				brsstrcpy((UDINT)p->user.dataBuffer, (UDINT)p->responseList.items[0]);
				bgSMRaiseDone(psm, 0);
			}

			if(ftpClientSingleCmdOnError(p)){
				bgSMRaiseError(psm, "got lower SM error", 0, 0);
			}
		break;
	}

	if(bgSMOnError(psm)){
		p->isErrorMultiCmd = p->userState;
		p->userState = 0;
		return;
	}

	if(bgSMOnDone(psm)){
		p->isDoneMultiCmd = p->userState;
		p->userState = 0;
	}
}
/*
########################################################################################
========================================================================================
FTP Connect command state machine:
*/
int ftpClientConnectOnDone(bgFtpClient_typ *p){
	return bgSMOnDone(&p->smCmdSocket);
}

int ftpClientConnectOnError(bgFtpClient_typ *p){
	return bgSMOnError(&p->smCmdSocket);
}

void ftpClientConnect(bgFtpClient_typ *p, int msgId)
{
DINT ret;
bgStateMachine_typ *psm = & p->smCmdSocket;

	if( msgId == BGSM_MSGID_INIT){
		bgSMReset(psm);
	}

    switch(bgSMCyclic(psm)){
        case 1:
			bgSMSetStateName(psm, "Connect-CreateSocket");

			if( bgSMIsStateInit(psm) ){
				p->cmdError = 0;
				p->cmdErrorCode = 0;
				p->isConnected = 0;
				/*create socket*/
				p->sock = socket(ETH_AF_INET, ETH_SOCK_STREAM, 0);

				if( p->sock == ERR_SOCKET ){
					bgSMRaiseError(psm, "socket create err", 0, EthGetError());
					break;
				}

				/*set non-blocking socket operation*/
				{
					UDINT arg = 1;
					ioctl(p->sock, ETH_FIONBIO, (UDINT)&arg);
				}

				/*reset select flags*/
				fd_zero((UDINT)&p->fdR);
				fd_zero((UDINT)&p->fdW);

				/*set time-out to 10ms*/
				p->timeOut.tv_sec = 0;
				p->timeOut.tv_usec = 1000 * 10;

				/*adjust my own timeout counters*/
				p->sockData_TimerCounter = 0;
				p->sockData_TimerTime = 10;
#if 0
/*bind not necessary*/
				/*bind client socket*/
				ret = bind(p->sock, (UDINT)&p->ftpClientAdrData, sizeof(p->ftpClientAdrData));
				if(ret == ERR_SOCKET){
					bgSMRaiseError(psm, "socket bind err", 0, EthGetError());
					break;
				}
#endif
			}

			/*connect to remote host*/
			ret = connect(p->sock, (UDINT)&p->ftpServerAdrCmd, sizeof(p->ftpServerAdrCmd) );

			if(ret == ERR_SOCKET){
				UINT errCode = EthGetError();
				if(errCode == ERR_ETH_INPROGRESS){
					/*next: wait connect to complete*/
					bgSMSetNextState(psm, bgSMGetState(psm) + 1);
				    break;
				}else
				if(errCode == ERR_ETH_ISCONN){
					/*it's connected -> done*/
					ERRxwarning(USER_ERROR_FTP, errCode, "connect()-alreadyOK!");
					bgSMRaiseDone(psm, 0);
					break;
				}
				else{
					bgSMRaiseError(psm, "socket connect err", 0, EthGetError());
					break;
				}
			}
			/*connected!*/
			ERRxwarning(USER_ERROR_FTP, ret, "connect()-OK-Quick!");
			bgSMRaiseDone(psm, 0);
		break;
		case 2:
			bgSMSetStateName(psm, "Connect-Connect");

			/*select waits for connection to complete*/
			fd_set(p->sock, (UDINT)&p->fdR);
			fd_set(p->sock, (UDINT)&p->fdW);
			ret = sock_select(32, (UDINT)&p->fdR, (UDINT)&p->fdW, 0L, (UDINT)&p->timeOut);

			if(ret == ERR_SOCKET){
				bgSMRaiseError(psm, "socket connect err", 0, EthGetError());
				break;
			}
/*
			DBG("connect: ret=%d, error=%d\n\r", ret, EthGetError());
*/
			if(ret == 0){
				if( p->sockData_TimerCounter >= p->sockData_TimerTime ){
					/*NOTES:
					- trying to figure out how does the select timeout works in B&R!
					- using EthGetError() here is not needed, just to see what comes back
					*/
					bgSMRaiseError(psm, "connect timeout", 0, EthGetError());
				}else{
					p->sockData_TimerCounter++;
				}
			}else{
				if( fd_isset(p->sock, (UDINT)&p->fdW) ){
					bgSMRaiseDone(psm, 0);
				}
			}
		break;
		default:
			/*unhandled state*/
			bgSMRaiseError(psm, "unknown state", 0, bgSMGetState(psm));
		break;
    }

	if( bgSMOnDone(psm)){
		ERRxwarning(USER_ERROR_FTP, 0, "connect()-OK!");
		p->isConnected = 1;
	}

	if( bgSMOnError(psm)){

	}
}
/*
========================================================================================
*/
void ftpClientMutliStateCmdErrorLog(bgFtpClient_typ *p){
char text[64];
	/*log error*/
	brsstrcpy((UDINT)&text[0], (UDINT)"Err: ");
	brsstrcat((UDINT)&text[0], (UDINT)&p->cmdSendBuf[0]);
    ERRxwarning(USER_ERROR_FTP, p->cmdErrorCode, &text[0]);
}
/*
########################################################################################
========================================================================================
FTP Login command state machine:
-return values:
*/
int ftpClientLoginOnDone(bgFtpClient_typ *p){
	return bgSMOnDone(&p->smFtpMultiCmd);
}

int ftpClientLoginOnError(bgFtpClient_typ *p){
	return bgSMOnError(&p->smFtpMultiCmd);
}
void ftpClientLogin(bgFtpClient_typ *p, int msgId)
{
bgStateMachine_typ *psm = &p->smFtpMultiCmd;

	if( msgId == BGSM_MSGID_INIT){
		bgSMReset(psm);
	}

    switch(bgSMCyclic(psm)){
        case 1:
			/*send USER name*/
			bgSMSetStateName(psm, "Login-Welcome");

			if( bgSMIsStateInit(psm) ){
				/*send request*/
				/*ftpClientSingleCmdInit(p, 0, ">name");*/
				ftpClientSingleCmdInit(p, 0, ">FTP");
			}

			/*recv response*/
			ftpClientSingleCmd(p);

			if(ftpClientSingleCmdOnDone(p)){
				bgSMSetNextState(psm, bgSMGetState(psm) + 1);
			}

			if(ftpClientSingleCmdOnError(p)){
				bgSMRaiseError(psm, "error in lower level SM", 0, 0);
			}
        break;
        case 2:
			/*send USER name*/
			bgSMSetStateName(psm, "Login-UserName");

			if( bgSMIsStateInit(psm) ){
				/*send request*/
				ftpClientSingleCmdInit(p, "USER  anonymous", "331");
			}

			/*recv response*/
			ftpClientSingleCmd(p);

			if(ftpClientSingleCmdOnDone(p)){
				bgSMSetNextState(psm, bgSMGetState(psm) + 1);
			}

			if(ftpClientSingleCmdOnError(p)){
				bgSMRaiseError(psm, "error in lower level SM", 0, 0);
			}
        break;
        case 3:
			/*send PASSWORD */
			bgSMSetStateName(psm, "Login-Password");

			if( bgSMIsStateInit(psm) ){
				/*send request*/
				ftpClientSingleCmdInit(p, "PASS  anonymous@", "230");
			}

			/*recv response*/
			ftpClientSingleCmd(p);

			if(ftpClientSingleCmdOnDone(p)){
				bgSMRaiseDone(psm, 0);
			}

			if(ftpClientSingleCmdOnError(p)){
				bgSMRaiseError(psm, "error in lower level SM", 0, 0);
			}
        break;
        default:
			/*unhandled state*/
			bgSMRaiseError(psm, "unknown state", 0, bgSMGetState(psm));
        break;
    }

	if( bgSMOnDone(psm) ){
		p->isLoggedIn = 1;
	}

	if( bgSMOnError(psm) ){
		ftpClientMutliStateCmdErrorLog(p);
	}

}
/*
########################################################################################
========================================================================================
FTP Logout command state machine:
-return values:
*/
int ftpClientLogoutOnDone(bgFtpClient_typ *p){
	return bgSMOnDone(&p->smFtpMultiCmd);
}

int ftpClientLogoutOnError(bgFtpClient_typ *p){
	return bgSMOnError(&p->smFtpMultiCmd);
}

void ftpClientLogout(bgFtpClient_typ *p, int msgId)
{
bgStateMachine_typ *psm = &p->smFtpMultiCmd;

	if( msgId == BGSM_MSGID_INIT){
		bgSMReset(psm);
	}

    switch(bgSMCyclic(psm)){
        case 1:
			/*send USER name*/
			bgSMSetStateName(psm, "Logout-Quit");

			if( bgSMIsStateInit(psm) ){
				/*send request*/
				ftpClientSingleCmdInit(p, "QUIT", "2??");
			}

			/*recv response*/
			ftpClientSingleCmd(p);

			if(ftpClientSingleCmdOnDone(p)){
				bgSMRaiseDone(psm, 0);
			}

			if(ftpClientSingleCmdOnError(p)){
				bgSMRaiseError(psm, "error in lower level SM", 0, 0);
			}
        break;
        default:
			/*unhandled state*/
			bgSMRaiseError(psm, "unknown state", 0, bgSMGetState(psm));
        break;
    }

	if(bgSMOnDone(psm)){
		p->isLoggedIn = 0;
	}

	if(bgSMOnError(psm)){
		p->isLoggedIn = 0;
		ftpClientMutliStateCmdErrorLog(p);
	}
}
/*
########################################################################################
========================================================================================
Lowest level state machine handles execution of a single FTP request/response messaging

ftpClientSingleCmdInit();
	- selects command to execute; init command state machine

ftpClientSingleCmd();
	- command execution state machine

ftpClientCmdCheckServerResponseCode()
	- command response check and verification

*/
void ftpClientSingleCmdInit(bgFtpClient_typ *p, char *cmd, char *expectedServerResponse){
int i;

	/*copy command string into send buffer*/
	p->cmdSendBuf[0]=0;
	if(cmd){
		brsstrcpy((UDINT)&p->cmdSendBuf[0], (UDINT)cmd);
		/*append string termination -> CRLF*/
		brsstrcat((UDINT)&p->cmdSendBuf[0], (UDINT)"\r\n");
	}

	/*define expected server response string?*/
	p->cmdExpectedServerResponse[0] = 0;	/*don't care*/
	if(expectedServerResponse){
		/*is expected server response code or string?*/
		if( *expectedServerResponse == '>'){
			i = 1;
			p->cmdExpectedServerResponseCodeOrString = 1;	/*string*/
		}else{
			i = 0;
			p->cmdExpectedServerResponseCodeOrString = 0;	/*code*/
		}
		bgStrCpyN(&p->cmdExpectedServerResponse[0], expectedServerResponse+i, FTPCLIENT_RESPONSECODE_LEN);
	}

	/*clr rcv buffer string*/
	memset(&p->cmdRecvBuf[0], 0, FTPCLIENT_CMDBUFSIZE);
#if 0
/*clear response lines*/
	/*init ptrs*/
	p->responseList.maxCount = CMD_RESPONSE_MAXLINES;
	p->responseList.lines[0] = &p->responseList.line0[0];
	p->responseList.lines[1] = &p->responseList.line1[0];
	p->responseList.lines[2] = &p->responseList.line2[0];
	p->responseList.lines[3] = &p->responseList.line3[0];
	p->responseList.lines[4] = &p->responseList.line4[0];

	/*clear all response lines*/
	for(i=0;i<CMD_RESPONSE_MAXLINES; i++){
		memset(p->responseList.lines[i], 0, CMD_RESPONSE_MAXLINELEN);
	}
	/*number of lines retrieved from the cmd buffer*/
	p->responseList.count = 0;
#endif
	/*number of lines retrieved from the cmd buffer*/
	p->responseList.itemCount = 0;

	/*reset command execution state machine*/
	bgSMReset(&p->smFtpCmd);
}

void ftpClientSingleCmd(bgFtpClient_typ *p){
DINT len;
DINT ret;
bgStateMachine_typ *psm = &p->smFtpCmd;

	/*state machine states*/
	switch( bgSMCyclic(psm) ){
		case 1:
          	/*send command request*/
			bgSMSetStateName(psm, "ftpSingleCmd");

			if(bgSMIsStateInit(psm)){
				/*check input conditions and paramters*/
				if( !p->isConnected ){
					bgSMRaiseError(psm, "not connected", 0, 0);
					break;
				}
				if( !p->cmdSendBuf[0]){
					/*nothing to send! receive only (i.e. welcome message just after connect()*/
					break;
				}

				/*send command to server*/
	         	len = strlen(&p->cmdSendBuf[0]);
	        	ret = send(p->sock, (UDINT)&p->cmdSendBuf[0], len, 0L);

	        	if(ret == ERR_SOCKET){
					bgSMRaiseError(psm, "send() error", 0, EthGetError());
					break;
	        	}

				/*remember the send length*/
				DBG("Single CMD send();Bytes=%d;[%s]\r\n", (int)ret, &p->cmdSendBuf[0]);
				p->sendLen = ret;
				return;
			}

	       	/*call receive (NON BLOCKING MODE!)*/
        	ret = recv(p->sock, (UDINT)&p->cmdRecvBuf[0],  FTPCLIENT_CMDBUFSIZE, 0L);

        	if(ret == ERR_SOCKET){
        		UINT errCode = EthGetError();
        		/*none blocking receive return this following value if data is not available yet*/
        		if( errCode == ERR_ETH_WOULDBLOCK ){
        			/*wait response*/
					return;
        		}

				/*recv error*/
				bgSMRaiseError(psm, "recv() error", 0, EthGetError());
				break;
        	}

			if(ret == 0){
				bgSMRaiseError(psm, "rx len=0", 0, 0);
				return;
			}

			/*receive is complete; store receive length & terminate rx buffer*/
			p->cmdRecvBuf[ret] = 0;
			DBG("Single CMD recv();Bytes=%d;[%s]\r\n", (int)ret, &p->cmdRecvBuf[0]);
			p->recvLen = ret;

			ret = ftpClientCmdCheckServerResponseCode(p);

			if( ret == 1)
				bgSMRaiseDone(psm, 0);

			if( ret == 2)
				bgSMRaiseError(psm, "server error response", 0, 0);

		break;
		default:
			/*unhandled state*/
			bgSMRaiseError(psm, "unknown state", 0, bgSMGetState(psm));
		break;
	}

	/*error event handler*/
	if(bgSMOnError(psm)){
		DBG("ftpClientSingleCmd - ERROR.\r\n");
	}

	/*done event handler*/
	if(bgSMOnDone(psm)){
		DBG("ftpClientSingleCmd - DONE.\r\n");
	}
}

int ftpClientSingleCmdOnError(bgFtpClient_typ *p)
{
	return bgSMOnError(&p->smFtpCmd);
}

int ftpClientSingleCmdOnDone(bgFtpClient_typ *p)
{
	return bgSMOnDone(&p->smFtpCmd);
}

/*
========================================================================================
FTP command response code is an ASCII line that looks like:
"xyz-response text<CR><LF>"
where x,y,z are numeric chars <0-9> followed by a '-' and the response text
- multiple lines per response are possible
- this function retrieves the response from the server, formats it into a list (array) of lines
and then searches each line for the user supplied code (res1,res2,res3)
- if res<x> is given as 0, it means don't care (see ftp spec)

*/
int ftpClientCmdCheckServerResponseCode(bgFtpClient_typ *p)
{
char serverResponseCode[3];
char *line;
int result;
int i;

	/*get server's response
	IMPORTANT:
	- note that data for ftpClientGetResponse() method is initilized within ftpClientSingleCmdInit()!
	- order of execution is like:
		init:
			ftpClientSingleCmdInit();
		cyclic:
			if( ftpClientSingleCmd() == DONE )
				if( ftpClientCmdCheckServerResponseCode() == OK )
					nextState;

	- therfore, the ftpClientGetResponse() shall be designed to operate in an incremenal mode: every time
	ftpClientSingleCmd() completes (data is available in the receive buffer) we should just add to the existing lines
	and not delete what we've received till that moment
	*/
	ftpClientGetResponse(p);

	/*final result of the ftpClientCmdCheckServerResponseCode() method:
	0 - response not found (not available -> wait)
	1 - response found (and it's ok; match with expected response)
	2 - response found (and it's not ok; error response from server)
	*/
	p->serverResponseCode = 0;

	/*anything to process!?*/
	if(!p->responseList.itemCount)
		return 0;

	/*check all received response lines every time (not necessary but it's easy to implement and it does not metter*/
	for(i=0; i<p->responseList.itemCount; i++){
		line = p->responseList.items[i];

		if(!p->cmdExpectedServerResponseCodeOrString){
			serverResponseCode[0]=*(line+0);
			serverResponseCode[1]=*(line+1);
			serverResponseCode[2]=*(line+2);

			result = 0;
			if( p->cmdExpectedServerResponse[0] != '?'){
				if(p->cmdExpectedServerResponse[0] == serverResponseCode[0])
					result++;
			}else
				result++;

			if( p->cmdExpectedServerResponse[1] != '?'){
				if(p->cmdExpectedServerResponse[1] == serverResponseCode[1])
					result++;
			}else
				result++;

			if( p->cmdExpectedServerResponse[2] != '?'){
				if(p->cmdExpectedServerResponse[2] == serverResponseCode[2])
					result++;
			}else
				result++;

			if( result >= 3)
				return 1;

			if( (serverResponseCode[0] == '4') || (serverResponseCode[0] == '5'))
				return 2;
		}else{
			result = bgStrFind(line, &p->cmdExpectedServerResponse[0], -1, -1);

			if(result >= 0)
				return 1;
		}
	}

	return 0;
}
/*
========================================================================================
*/
void ftpClientGetResponse(bgFtpClient_typ *p){
int i;
char *src;

	/*ptr to rcv buffer*/
	src = &p->cmdRecvBuf[0];
	p->responseList.src = src;
	bgStringListLines(&p->responseList);

	DBG("Received Cmd Response: lines=%d\r\n", p->responseList.itemCount);
	for(i=0;i<p->responseList.itemCount;i++){
		DBG("Line[%d]=%s\r\n", i, p->responseList.items[i]);
	}

}

int readline(char *src, char *dest, int maxLength){
/*
return: >= 0 (length of the line including CRLF)
return: -1 (no line read)
*/
int lineLen;
char *cPtr;

	lineLen = 0;
	cPtr = src;
	while(maxLength--){

		if( (*cPtr == 0x0D) || ( *cPtr == 0x0A) ){

			lineLen++;
			cPtr++;

			if( (*cPtr == 0x0D) || ( *cPtr == 0x0A) ){
				lineLen++;
			}

			memcpy(dest, src, lineLen);
			*(dest+lineLen+1)= 0;
			return lineLen;
		}

		if( *cPtr == 0 )
			return -1;

		lineLen++;
		cPtr++;
	}

	return -1;
}

/*
========================================================================================
*/
int ftpClientCmdMultiOnDone(bgFtpClient_typ *p, int cmdId)
{
/*generate CmdIsDone signal (1 shoot)*/
	if( p->isDoneMultiCmd == cmdId ){
		p->isDoneMultiCmd = 0;
		return 1;
	}else
		return 0;
}

int ftpClientMultiCmdOnError(bgFtpClient_typ *p, int cmdId){
/*generate CmdIsError signal (1 shoot)*/
	if( p->isErrorMultiCmd == cmdId ){
		p->isErrorMultiCmd = 0;
		return 1;
	}else
		return 0;
}

/*
========================================================================================
*/
void bgFtpClientConnectAndLogin(bgFtpClient_typ *p, char *ethernetDevice, char *serverIp)
{
unsigned long ipAddrClient;

    /*set server ip address and ports to use*/
    /*  21 - standard FTP command port
        20 - standard FTP data port
    */
	setSocketAddressData(&p->ftpServerAdrCmd, serverIp, 21);
	setSocketAddressData(&p->ftpClientAdrData, "", ETH_INADDR_ANY);

	/*retrieve own ip address*/
	p->CfgIPAddr_1.enable = 1;
	p->CfgIPAddr_1.pDevice = (UDINT)ethernetDevice;
	p->CfgIPAddr_1.pIPAddr = (UDINT)&p->CfgIPAddrString[0];
	p->CfgIPAddr_1.Len = 16;
	CfgGetIPAddr(&p->CfgIPAddr_1);

	ipAddrClient = inet_addr( (unsigned long) &p->CfgIPAddrString[0]);

	/*store ip address in an easy format for later use; see PORT command*/
	p->ipAddr[3]= (ipAddrClient>>24)&0xFF;
	p->ipAddr[2]= (ipAddrClient>>16)&0xFF;
	p->ipAddr[1]= (ipAddrClient>>8)&0xFF;
	p->ipAddr[0]= (ipAddrClient)&0xFF;

	p->cmdError = 0;
	p->cmdErrorCode = 0;
	p->isConnected = 0;
    p->user.connectRequest = 1;
}
/*
========================================================================================
*/
int bgFtpClientIsLoggedIn(bgFtpClient_typ *p)
{
    return p->isLoggedIn;
}

/*
========================================================================================
*/
void bgFtpClientDisconnect(bgFtpClient_typ *p)
{
    p->user.disconnectRequest = 1;
}
/*
========================================================================================
*/
int bgFtpClientIsConnected(bgFtpClient_typ *p)
{
    return p->isConnected;
}
/*
========================================================================================
*/
int bgFtpClientIsError(bgFtpClient_typ *p)
{
    return p->cmdError;
}

int ftpClientIncrDataPort(bgFtpClient_typ *p){

	if( !p->dataPort){
		p->dataPort = 190;
	}

	if(p->dataPort>=190)
		p->dataPort++;

	if(p->dataPort>=200)
		p->dataPort = 190;

	return p->dataPort;
}
/*
========================================================================================
*/
void ftpClientCmdTextPort(bgFtpClient_typ *p, char *textBuffer)
{
/*
	bgsprintf(textBuffer, "PORT 192,168,1,6,4,%d", p->dataPort);
*/
	sprintf2(textBuffer, "PORT %d,%d,%d,%d,4,%d", p->ipAddr[0], p->ipAddr[1], p->ipAddr[2], p->ipAddr[3], p->dataPort);
}
/*
========================================================================================
*/
int ftpClientDataServerOnError(bgFtpClient_typ *p)
{
	return bgSMOnError(&p->smDataSocket);
}

int ftpClientDataServerOnDone(bgFtpClient_typ *p)
{
	return bgSMOnDone(&p->smDataSocket);
}

void ftpClientDataServer(bgFtpClient_typ *p, int msgId)
{
bgStateMachine_typ *psm = &p->smDataSocket;

    /*init data socket (listen)*/
	if( (msgId == BGSM_MSGID_INIT) ){
		bgSMReset(psm);
		p->sockData_TimerTime = 10;
		p->sockData_TimerCounter = 0;
		p->recvLenData = 0;
		p->sendLenData = 0;
		return;
	}

    /*close data socket (listen stop)*/
	if( msgId == 2){
		/*command socket is telling us to receive data from server
		after this event, keep receiving until we don't get any data
		for a certain period of time or the remote host closes the
		connection
		*/
		p->sockData_Timer = 1;
		p->sockData_TimerTime = 20;
		p->sockData_TimerCounter = 0;
		return;
	}

    /*close data socket now!*/
	if( msgId == 3){
		/*command socket is telling us to immediately close data socket
		*/
		bgSMSetNextState(psm, 3);
		return;
	}

	switch(bgSMCyclic(psm)){
		case 1:
			bgSMSetStateName(psm, "DataPort-Init");
			if(bgSMIsStateInit(psm)){
				p->sockData_Timer = 0;

				p->TCPserv_1.enable = 1;            /* enables the FUB */
	    		p->TCPserv_1.porta = 4*256 + p->dataPort;           	/* port number of the server */
	    		TCPserv(&p->TCPserv_1);				/* makes a connection with the clients */

	    		p->TCPrecv_1.enable = 1;           	/* enables the FUB */
				p->rxDataBuff = 0;
				p->recvLenData = 0;
				p->TCPrecv_1.mxbuflng = 10000;		/* size of the buffer should be > 8192*/
    			TMP_alloc (p->TCPrecv_1.mxbuflng, (void**)&p->rxDataBuff);   /*allocate memory for data rx*/
	    		p->TCPrecv_1.buffer = (UDINT)p->rxDataBuff; /* address of the buffer */

	    		p->TCPclose_1.enable = 1;                  /* enables the FUB */

				DBG("data port open\r\n");
				break;

			}

    		TCPserv(&p->TCPserv_1);					/*listen for a server connection request*/

			/*server connection accepted*/
			if(p->TCPserv_1.status == 0){
				/*NOTE: data port is ready if either connection is accepted or if waiting for connection*/
				DBG("datasocket - connected\r\n");
				p->isDataPortReady = 1;
 				bgSMSetNextState(psm, bgSMGetState(psm) + 1);
				break;
			}

			/*waiting for connection || pNA is busy*/
			if( (p->TCPserv_1.status == 0xFFFF) || (p->TCPserv_1.status == 14893) ){
				DBG("datasocket - waiting connection\r\n");
				p->isDataPortReady = 1;
				break;
			}

			DBG("datasocket - error=%d\r\n", p->TCPserv_1.status);

			bgSMRaiseError(psm, "TCPserv() error", 0, p->TCPserv_1.status);
		break;
		case 2:
			bgSMSetStateName(psm, "DataPort-Recv");
			/* recv in progress*/
   			p->TCPrecv_1.cident = p->TCPserv_1.cident;    /* copy serv() Id to recv() */
           	TCPrecv(&p->TCPrecv_1);

			/*recv timer*/
		p->sockData_TimerCounter++;
            if(p->sockData_Timer && (p->TCPrecv_1.status == 0xFFFF)){
    			/*p->sockData_TimerCounter++;*/
				DBG("data port recv() busy; counter=%d\r\n", p->sockData_TimerCounter);
            }

            if(p->TCPrecv_1.status == 0){
				/*test only; inc receive counter*/
				p->counter++;

				/*in case data arrives->copy data to user buffer*/
				if(p->TCPrecv_1.rxbuflng != 0){

					if(p->user.dataBufferLength < (p->recvLenData + p->TCPrecv_1.rxbuflng) ){
						DBG("!!!! rxBufferOverflow rxLen=%d > rxBufferSize=%d!!!!\r\n", (int)(p->recvLenData + p->TCPrecv_1.rxbuflng), (int)p->user.dataBufferLength);
						DBG("!!!! INCREASE USER RX BUFFER SIZE !!!!\r\n");
						/*user supplied buffer is too small!!!*/
						bgSMRaiseError(psm, "Data Buffer Overflow!", 0, bgSMGetState(psm));
						break;
					}

					memcpy( (char*)(p->user.dataBuffer + p->recvLenData), p->rxDataBuff, p->TCPrecv_1.rxbuflng);
					p->recvLenData += p->TCPrecv_1.rxbuflng;

					p->sockData_TimerCounter = 0;
				}
				else{
					/*Status == 0 && rxLengt == 0 -> remote peer has closed the connection!!!*/
					bgSMSetNextState(psm, bgSMGetState(psm) + 1);
				}
            }
			else
			if(p->sockData_TimerCounter >= p->sockData_TimerTime){
				/*if receive timer expires, close data socket*/
				bgSMSetNextState(psm, bgSMGetState(psm) + 1);
			}

			DBG("data recv(); rxLen=%d, rxStatus=%d, timer=%d \r\n",
				(int)p->TCPrecv_1.rxbuflng, (int)p->TCPrecv_1.status, (int)p->sockData_TimerCounter);
		break;
		case 3:
			bgSMSetStateName(psm, "DataPort-Close");
   			p->TCPclose_1.cident = p->TCPserv_1.cident;    	/* copy the  Ident number */
            TCPclose(&p->TCPclose_1);          /* set the socket free */

			if(p->TCPclose_1.status == 0){
				p->isDataPortReady = 0;
				p->sockData_Timer = 0;

				/*terminate rx buffer with 0 -> for strings*/
				p->user.dataBuffer[p->recvLenData] = 0;

				bgSMRaiseDone(psm, 0);
			}

			if( p->rxDataBuff ){
				p->rxDataBuff = 0;
				TMP_free (p->TCPrecv_1.mxbuflng, (void**)p->rxDataBuff);
			}
		break;
		default:
			/*unhandled state*/
			bgSMRaiseError(psm, "unknown state", 0, bgSMGetState(psm));
		break;
	}

	if(bgSMOnError(psm)){
		p->TCPclose_1.cident = p->TCPserv_1.cident;    	/* copy the  Ident number */
	    TCPclose(&p->TCPclose_1);          				/* set the socket free */
		p->isDataPortReady = 0;

		if( p->rxDataBuff ){
			p->rxDataBuff = 0;
			TMP_free (p->TCPrecv_1.mxbuflng, (void**)p->rxDataBuff);
		}
		/*raise error again for cmd level state machine*/
		bgSMRaiseError(psm, "Data Server Error", 0, 0);
 	}

	if(bgSMOnDone(psm)){

	}
}
/*
========================================================================================
*/
void swapBytesInShort(unsigned short *value)
{

union{
	unsigned short 	shortValue;
	unsigned char	bytes[2];
}swapValue;

unsigned char tempByte;

	swapValue.shortValue = *value;
	tempByte = swapValue.bytes[0];
	swapValue.bytes[0] = swapValue.bytes[1];
	swapValue.bytes[1] = tempByte;
	*value = swapValue.shortValue;
}
/*
========================================================================================
*/
void setSocketAddressData(ETH_sockaddr_typ *adrData, char *hostIpAddressString, unsigned short hostPort)
{

	unsigned short sin_family;
	unsigned short family;
	unsigned short length;
	unsigned short port;

	family = ETH_AF_INET;
	length = sizeof(ETH_sockaddr_typ);
	sin_family = (family << 8) + length;

	adrData->sin_family = sin_family;
	port = hostPort;
	swapBytesInShort(&port);
	adrData->sin_port = port;
	if( strlen(hostIpAddressString) < 8)
		adrData->sin_addr = ETH_INADDR_ANY;
	else
		adrData->sin_addr = inet_addr( (unsigned long) hostIpAddressString);
	adrData->sin_zero[0]=0;
	adrData->sin_zero[1]=0;
	adrData->sin_zero[2]=0;
	adrData->sin_zero[3]=0;
	adrData->sin_zero[4]=0;
	adrData->sin_zero[5]=0;
	adrData->sin_zero[6]=0;
	adrData->sin_zero[7]=0;
}
/*
========================================================================================
========================================================================================
========================================================================================
========================================================================================
*/
/*EOF*/
```

### bgBitUtilities.c
```c
#include <bur/plctypes.h>
#ifndef _BG_BITUTILS_C
#define _BG_BITUTILS_C

#include <bur/plctypes.h>

void bgBitSetUDINT(UDINT* dest,  UINT bitIndex, BOOL bitValue)
{
	UDINT mask = 0x1;
	UDINT current = *dest;

	mask <<= bitIndex;

	if(!(bitValue && 0x1) ){
		mask = ~(mask);
		current &= mask;
	}else{
		current |= mask;
	}

	*dest = current;
}

void bgBitSetUINT(UINT* dest,  UINT bitIndex, BOOL bitValue)
{
	UINT mask = 0x1;
	UINT current = *dest;

	mask <<= bitIndex;

	if(!(bitValue && 0x1) ){
		mask = ~(mask);
		current &= mask;
	}else{
		current |= mask;
	}

	*dest = current;
}

void bgBitSetUSINT(USINT* dest,  UINT bitIndex, BOOL bitValue)
{
	USINT mask = 0x1;
	USINT current = *dest;

	mask <<= bitIndex;

	if(!(bitValue && 0x1) ){
		mask = ~(mask);
		current &= mask;
	}else{
		current |= mask;
	}

	*dest = current;
}
#endif
//eof
```

### bgBufMemAlloc.h
```c
/**\file: bgBufMemAlloc.h
*Buffer memory (user supplied memory) simple allocation methods.
*/
#ifndef _BG_BUFMEMALLOC_H
#define _BG_BUFMEMALLOC_H

/**
\def BGBUFMEMALLOC_MAX_BLOCKS
Defines maximum number of items within the list of memory blocks.
Used for data object: \link bgBufMemAlloc_typ \endlink
*/
#define BGBUFMEMALLOC_MAX_BLOCKS	16

/**
\struct bgBufMemAlloc_typ
Data object that holds information about simple memory allocation method.\n
In a deeply embedded systems, memory allocation is rather uncommon practice. However,
there are situations (i.e. networking) where certain, simplified "mem allocation" scheme
is rather useful.\n
This data object and associated methods implement memory allocation scheme that uses
user suppllied memory buffer as the "source memory".
*/
typedef struct bgBufMemAlloc_typ{
	char* pBufMem;			/**<Input: User supplied memory buffer*/
	int lengthBufMemBytes; 	/**<Input: Lenght (bytes) of the user supplied memory buffer*/

    int countMaxBlocks;		/**<Input(const): Max number of mem blocks*/
    int countUsedBlocks;	/**<Output: Number of currently allocated blocks*/
    int lengthUsedMemBytes;	/**<Output: Total length (bytes) of currently allocated memory*/

    struct bgBufMemBlock_typ{
		int 	used;			/**<I/O: 0-block not used; 1-block is used*/
        char*   pMemBlock;		/**<Output: Ptr to the mem block*/
        int     lengthMemBlockBytes;	/**<Input: Size (bytes) of the mem block*/
    }memBlock[BGBUFMEMALLOC_MAX_BLOCKS];

}bgBufMemAlloc_typ;

/**
Init method for data object: \link bgBufMemAlloc_typ \endlink
\param p Ptr to data object: \link bgBufMemAlloc_typ \endlink
\param pBufMem Ptr to user supplied memory buffer
\param lengthBufMemBytes Size of the user supplied memory buffer
<b>IMPORTANT: </b>This method <b>must be always</b> called first for the associated data object!\n

*/
void bgBufMemAllocInit(bgBufMemAlloc_typ* p, char* pBufMem, int lengthBufMemBytes);

/**
Method for data object: \link bgBufMemAlloc_typ \endlink\n
Creates / allocates memory block of size (sizeMemBlock)
\param p Ptr to data object: \link bgBufMemAlloc_typ \endlink
\param blockSize Requested memory block size
\param pMemBlock Address to store the pointer to newly allocated mem block
\param sizeMemBlock Address to store the size of the newly allocated mem block
\return Id for the allocated mem block (0 to (BGBUFMEMALLOC_MAX_BLOCKS-1))
*/
int bgBufMemAllocCreateBlock(bgBufMemAlloc_typ* p, int blockSize, char** pMemBlock, int* sizeMemBlock);

/**
Method for data object: \link bgBufMemAlloc_typ \endlink\n
Give the memblock Id, returns the memory and size of the requesed memblock
\param p Ptr to data object: \link bgBufMemAlloc_typ \endlink
\param blockId Id of the mem block previosly allocated using \link bgBufMemAllocCreateBlock \endlink
\param blockSize Address to store the size of the newly allocated mem block
\return Address of the newly allocated mem block or NULL (in case the blockId is invalid)
*/
char* bgBufMemAllocGetBlockPtr(bgBufMemAlloc_typ* p, int blockId, int* blockSize);

/*
##################################################################################
String heap
##################################################################################
*/

/**
\struct bgStringHeap_typ
Data object that holds information about simple memory allocation method for strings.\n
In a deeply embedded systems, dynamic string memory allocation is rather uncommon practice.
However, there are situations (i.e. networking) where certain, simplified dynamic allocation
scheme for storing variable lenght strings is rather useful.\n
This data object and associated methods implement dynamic memory allocation scheme for
strings that uses user suppllied memory buffer as a memory to store variable length strings.
*/
typedef struct bgStringHeap_typ{
	char* pMemStart;	/**<Start of the user supplied memory buffer*/
	int	memSize;		/**<Size (bytes) of the user supplied memory buffer*/
	char* pMemCurrent;	/**<Ptr to the current free memory location within the (pMemStart)*/
	int memFree;		/**<Size (bytes) of still available / free memory*/
}bgStringHeap_typ;

/**
Method for data object: \link bgStringHeap_typ \endlink\n
Creates / allocates memory block of size (sizeMemBlock)
\param pHeap Ptr to data object: \link bgStringHeap_typ \endlink
\param pHeapMem User supplied memory that will be used for storage of dynamic strings
\param memSize Size of the user supplied memory
\return Ptr to the start of memory (same as pHeapMem) or NULL if error
<b>IMPORTANT: </b>This method <b>must be always</b> called first for the associated data object!\n
*/
char* bgStringHeapInit(bgStringHeap_typ* pHeap, char* pHeapMem, int memSize);

/**
Method for data object: \link bgStringHeap_typ \endlink\n
Stores given string (pStr) to the string heap memory. Returns ptr to the stored string.
\param pHeap Ptr to data object: \link bgStringHeap_typ \endlink
\param pStr String to store on the string heap
\return Ptr to string stored on the heap or NULL if error (not enough space)
*/
char* bgStringHeapAddString(bgStringHeap_typ* pHeap, char* pStr);

#endif
```

### bgDataStructures.h
```c
/**\file: bgDataStructures.h
*Common data structures. (stack, list, tree, etc.)
*/
#ifndef _BG_DATASTRUCTURES_H
#define _BG_DATASTRUCTURES_H

/*
##################################################################################
Stack
##################################################################################
*/
/**
\def BGSTACK_DEPTH_MAX
Defines maximum number of items on the stack (stack depth)
*/
#define BGSTACK_DEPTH_MAX	64

/**
\struct bgStack_typ
Data object that represents a stack (of ptr-s)\n
*/
typedef struct bgStack_typ{
    int index;	/**<Position of the next empty location on the stack.*/
	char* data[BGSTACK_DEPTH_MAX]; /**<Array that holds the stack.*/
}bgStack_typ;

/**
Method for data object \link bgStack_typ \endlink\n
This method must be called first, prior from calling any other method related to this data object.
\param stack Ptr to data object: (\link bgStack_typ \endlink)
*/
void bgStackInit(bgStack_typ* stack);

/**
Method for data object \link bgStack_typ \endlink\n
Push item to the stack.
\param stack Ptr to data object: (\link bgStack_typ \endlink)
\param data Ptr that will be pushed / stored on the stack.
\return Same ptr that is pushed to the stack (data) or NULL if stack if full.
*/
char* bgStackPush(bgStack_typ* stack, char* data);

/**
Method for data object \link bgStack_typ \endlink\n
Pop (retrive) item from the stack.
\param stack Ptr to data object: (\link bgStack_typ \endlink)
\return Ptr that represent item from the stack (or NULL if none)
*/
char* bgStackPop(bgStack_typ* stack);

/**
Method for data object \link bgStack_typ \endlink\n
Retrieve top item (ptr) from the stack wo. removing it from the stack.
\param stack Ptr to data object: (\link bgStack_typ \endlink)
\return Ptr that represent top item from the stack (or NULL if none)
*/
char* bgStackPeek(bgStack_typ* stack);

/**
Method for data object \link bgStack_typ \endlink\n
Return number of items stored on the stack.
\param stack Ptr to data object: (\link bgStack_typ \endlink)
\return Number of items on the stack.
*/
int bgStackGetItemCount(bgStack_typ* stack);

/*
##################################################################################
Tree  of Nodes (Each nodes has lf,rt,up,dw connections - 4C(onnections) nodes)
##################################################################################
*/

/**
\struct bgTree4CNode_typ
Data object represents a node w. 4-way connections (left, right, up, down)
*/
typedef struct bgTree4CNode_struct{
	int used;				/**<0-not used; 1-used*/
	int id;					/**<Node Id (unique identifier); 0 to (nodeCountMax - 1)*/
	int nodeCountMax;		/**<Max number of nodes (depends on the available memory)*/
	struct bgTree4CNode_struct*	up;	/**<Link (ptr) to the up node (or 0 if none)*/
	struct bgTree4CNode_struct*	dw; /**<Link (ptr) to the down node (or 0 if none)*/
	struct bgTree4CNode_struct*	rt; /**<Link (ptr) to the right node (or 0 if none)*/
	struct bgTree4CNode_struct*	lf; /**<Link (ptr) to the left node (or 0 if none)*/
	int dataType;			/**<Type of data node is holding*/
	int dataValue;			/**<Local data storage; used for simple, scalar types (int, bool)*/
	char* data;				/**<Ptr to data storage (string type, etc.)*/
}bgTree4CNode_typ;

/**
\struct bgTree4C_typ
Data object holds a tree of 4-way nodes.
*/
typedef struct bgTree4C_typ{
	int nodeCountUsed;			/**<Number of used nodes*/
	int nodeCountMax;			/**<Max number of nodes*/
	bgTree4CNode_typ* nodes;	/**<Ptr to user supplied buffer / memory for node storage*/
}bgTree4C_typ;

/**
Method for data object \link bgTree4C_typ \endlink\n
This method must be called first, prior from calling any other method related to this data object.
\param tree Ptr to data object: (\link bgTree4C_typ \endlink)
\param treeMem Ptr to user supplied buffer / memory of nodes
\param treeMemSize Size (bytes) of user supplied buffer / memory of nodes

*/
void bgTree4CInit(bgTree4C_typ* tree, char* treeMem, int treeMemSize);

void bgTree4CNodeClr(bgTree4CNode_typ* node);

bgTree4CNode_typ* bgTree4CNodeCreate(bgTree4C_typ* tree);
void bgTree4CNodeDelete(bgTree4C_typ* tree, bgTree4CNode_typ* node);

bgTree4CNode_typ*  bgTree4CNodePreviousLevel(bgTree4CNode_typ* node1);
bgTree4CNode_typ* bgTree4CGetNextNodeRtDw(bgTree4CNode_typ* node1);
bgTree4CNode_typ* bgTree4CGetNextNodeDw(bgTree4CNode_typ* node1);
bgTree4CNode_typ*  bgTree4CGetRootNode(bgTree4C_typ* tree);
bgTree4CNode_typ* bgTree4CNodeGetNextLf(bgTree4CNode_typ* node);

void bgTree4CNodeAddDw(bgTree4CNode_typ* node1, bgTree4CNode_typ* node2);
void bgTree4CNodeAddRt(bgTree4CNode_typ* node1, bgTree4CNode_typ* node2);
int bgTree4CNodeAppendToDwEnd(bgTree4CNode_typ* node1, bgTree4CNode_typ* node2);
int bgTree4CNodeAppendToRtEnd(bgTree4CNode_typ* node1, bgTree4CNode_typ* node2);
int	bgTree4CNodeInsertRt(bgTree4CNode_typ* node1, bgTree4CNode_typ* node2);
int	bgTree4CNodeInsertLf(bgTree4CNode_typ* node1, bgTree4CNode_typ* node2);

void bgTree4CNodeSetDataType(bgTree4CNode_typ* node, int dataType);
void bgTree4CNodeSetDataValue(bgTree4CNode_typ* node, int dataVal);
void bgTree4CNodeSetDataPtr(bgTree4CNode_typ* node, char* data);

int bgTree4CGetCountFreeNodes(bgTree4C_typ* tree);

void bgTree4CPrint(bgTree4C_typ* tree);

#endif
```

### bgPVLogger.c
```c
/********************************************************************
 * COPYRIGHT -- belgor
 ********************************************************************
 * Package: bglib
 * File: bgPVLogger.c
 * Author: goran
 * Created: October 13, 2011
 *******************************************************************/

#include <bur/plctypes.h>
//#ifdef _DEFAULT_INCLUDES
#include <AsDefault.h>

/**
 Simple logging.
 Set to 0 when simple log is not needed
 To view this log, open Automation Studio  watch window and insert below defined
 logxx variable.
 Most recent log entry is always on the top (index 0)
 */
#if 1
#include "bgsprintf.h"
#include "bgsprintf.c"
#include "bgstring.h"
#include "bgstring.c"

typedef struct bgPVLogger_typ
{
	int initOk;
	char* logbuf;
	int entryCount;
	int entryLen;
}bgPVLogger_typ;

static void bgPVLoggerInit(bgPVLogger_typ* p, char* logbuf, int logEntryCount, int logEntryLen)
{
	if(!logbuf || !logEntryCount || !logEntryLen)
		return;

	p->logbuf = logbuf;
	p->entryCount = logEntryCount;
	p->entryLen = logEntryLen;
	p->initOk = 1;
}

static void shiftlog(bgPVLogger_typ* p)
{
int ii;
	if(!p || !p->initOk)
		return;

	for(ii=(p->entryCount-2); ii>=0; ii--){
		bgStrCpyN(&p->logbuf[(ii+1) * p->entryLen], &p->logbuf[ii * p->entryLen], p->entryLen);
	}
}

#define DBG(loggerInstance, format, args...)	shiftlog(&loggerInstance); bgsnprintf(&loggerInstance.logbuf[0], loggerInstance.entryLen, format, ## args);
#define DBGINIT(loggerInstance,  logbuf, logEntryCount, logEntryLen) bgPVLoggerInit(&loggerInstance, &logbuf[0][0], logEntryCount, logEntryLen);

#else

#define DBG(format, args...)   ;

#endif

//#endif
```

### bgringbuffer.h
```c
/*
File:
bgRingBuffer.c

About:
------
- ring buffer implementation

*/
#ifndef _BG_RINGBUFFER_H
#define _BG_RINGBUFFER_H

#define BG_DEBUG_FORMAT_FILENAME	0x1
#define BG_DEBUG_FORMAT_FUNCTION	0x2
#define BG_DEBUG_FORMAT_TIMESTAMP	0x4
#define BG_DEBUG_FORMAT_LEVEL		0x8

/*
Public data types:
-----------------
*/
typedef struct bgRingBuffer_typ{

    int     bufSize;
    int     init;
    int     overrun;
    int     dbgLevel;
    int     dbgFormat;

    char    *ptrCircularBufferBegin;
    char    *ptrCircularBufferEnd;

    char    *ptrDataIn;
    char    *ptrDataOut;

}bgRingBuffer_typ;

/*
Public functions:
-----------------
*/
/*
- copy max. destSize bytes of data from the ring buffer to *destination
*/
int bgRingBuffGet(bgRingBuffer_typ *rb, char *destination, int destSize);

/*
- copy *sourceString (null terminated c-style string) into the ring buffer
*/
void bgRingBuffPutString(bgRingBuffer_typ *rb, char *sourceString);

/*
- before RingBuffer can be used data buffer of size destinationBufferSize must be defined
(use allocated or _LOCAL/_GLOBAL space)
*/
void bgRingBuffInit(bgRingBuffer_typ *rb, char *destination, int destinationBufferSize);

/*
- debug specific function for entering data into the ring buffer
*/
void bgRingBuffPutDbgInfo(bgRingBuffer_typ *rb, char *file, char *function, unsigned int level, unsigned int context, char *format, ...);

/*
- put formated message (i.e. printf) into the ring buffer
*/
//void bgRingBuffPrintf(bgRingBuffer_typ *rb, char *format, ...);

#endif
```
